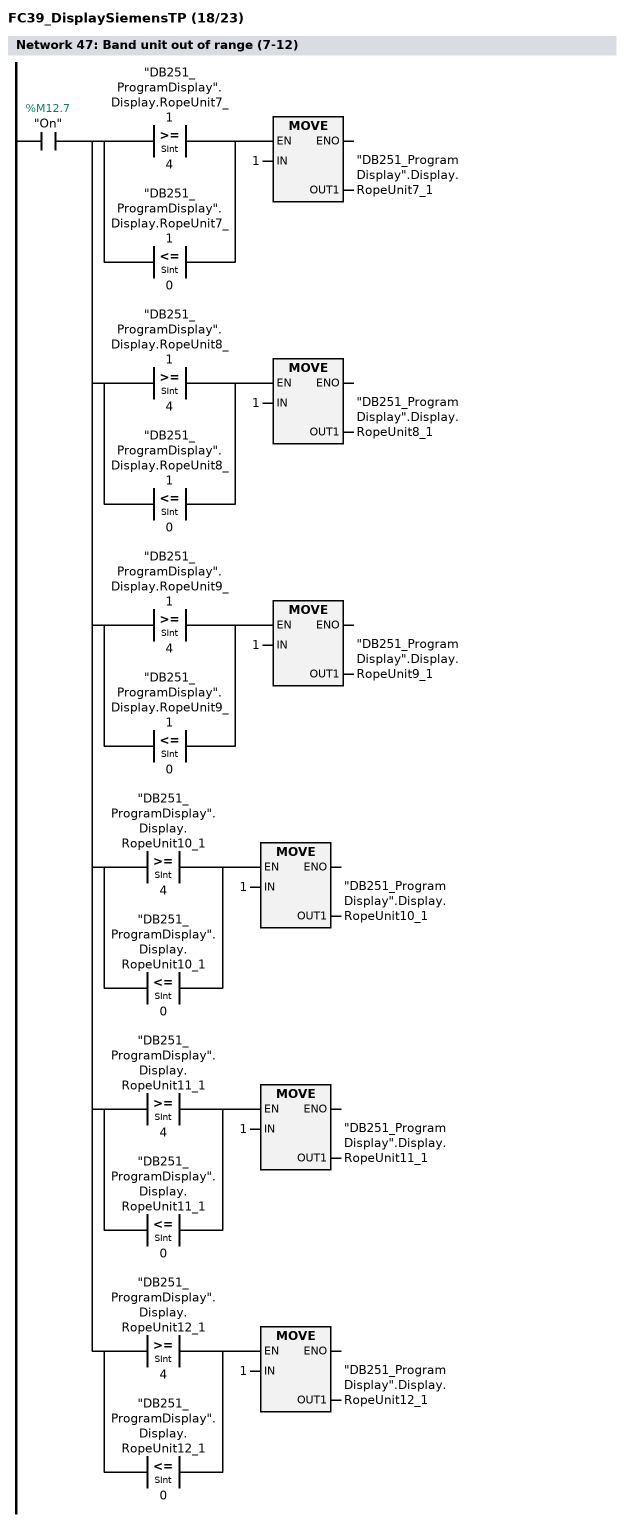
   RUNG wire#powerrail
      Contact( "On" )
      wire#w1
      { S7_Templates := "SrcType := SInt" } GE_Contact(in1 := "DB251_ProgramDisplay".Display.RopeUnit7_1, in2 := 4)
      wire#w2
      { S7_GenerateENO := "TRUE" } Move(in := 1, out1 => "DB251_ProgramDisplay".Display.RopeUnit7_1)
   END_RUNG
   RUNG wire#w1
      { S7_Templates := "SrcType := SInt" } LE_Contact(in1 := "DB251_ProgramDisplay".Display.RopeUnit7_1, in2 := 0)
   END_RUNG wire#w2
   RUNG wire#w1
      { S7_Templates := "SrcType := SInt" } GE_Contact(in1 := "DB251_ProgramDisplay".Display.RopeUnit8_1, in2 := 4)
      wire#w3
      { S7_GenerateENO := "TRUE" } Move(in := 1, out1 => "DB251_ProgramDisplay".Display.RopeUnit8_1)
   END_RUNG
   RUNG wire#w1
      { S7_Templates := "SrcType := SInt" } LE_Contact(in1 := "DB251_ProgramDisplay".Display.RopeUnit8_1, in2 := 0)
   END_RUNG wire#w3
   RUNG wire#w1
      { S7_Templates := "SrcType := SInt" } GE_Contact(in1 := "DB251_ProgramDisplay".Display.RopeUnit9_1, in2 := 4)
      wire#w4
      { S7_GenerateENO := "TRUE" } Move(in := 1, out1 => "DB251_ProgramDisplay".Display.RopeUnit9_1)
   END_RUNG
   RUNG wire#w1
      { S7_Templates := "SrcType := SInt" } LE_Contact(in1 := "DB251_ProgramDisplay".Display.RopeUnit9_1, in2 := 0)
   END_RUNG wire#w4
   RUNG wire#w1
      { S7_Templates := "SrcType := SInt" } GE_Contact(in1 := "DB251_ProgramDisplay".Display.RopeUnit10_1, in2 := 4)
      wire#w5
      { S7_GenerateENO := "TRUE" } Move(in := 1, out1 => "DB251_ProgramDisplay".Display.RopeUnit10_1)
   END_RUNG
   RUNG wire#w1
      { S7_Templates := "SrcType := SInt" } LE_Contact(in1 := "DB251_ProgramDisplay".Display.RopeUnit10_1, in2 := 0)
   END_RUNG wire#w5
   RUNG wire#w1
      { S7_Templates := "SrcType := SInt" } GE_Contact(in1 := "DB251_ProgramDisplay".Display.RopeUnit11_1, in2 := 4)
      wire#w6
      { S7_GenerateENO := "TRUE" } Move(in := 1, out1 => "DB251_ProgramDisplay".Display.RopeUnit11_1)
   END_RUNG
   RUNG wire#w1
      { S7_Templates := "SrcType := SInt" } LE_Contact(in1 := "DB251_ProgramDisplay".Display.RopeUnit11_1, in2 := 0)
   END_RUNG wire#w6
   RUNG wire#w1
      { S7_Templates := "SrcType := SInt" } GE_Contact(in1 := "DB251_ProgramDisplay".Display.RopeUnit12_1, in2 := 4)
      wire#w7
      { S7_GenerateENO := "TRUE" } Move(in := 1, out1 => "DB251_ProgramDisplay".Display.RopeUnit12_1)
   END_RUNG
   RUNG wire#w1
      { S7_Templates := "SrcType := SInt" } LE_Contact(in1 := "DB251_ProgramDisplay".Display.RopeUnit12_1, in2 := 0)
   END_RUNG wire#w7
   // the same network as SCL:
   IF "On" AND (("DB251_ProgramDisplay".Display.RopeUnit7_1 >= 4) OR ("DB251_ProgramDisplay".Display.RopeUnit7_1 <= 0)) THEN
       "DB251_ProgramDisplay".Display.RopeUnit7_1 := 1;
   END_IF;
   IF "On" AND (("DB251_ProgramDisplay".Display.RopeUnit8_1 >= 4) OR ("DB251_ProgramDisplay".Display.RopeUnit8_1 <= 0)) THEN
       "DB251_ProgramDisplay".Display.RopeUnit8_1 := 1;
   END_IF;
   IF "On" AND (("DB251_ProgramDisplay".Display.RopeUnit9_1 >= 4) OR ("DB251_ProgramDisplay".Display.RopeUnit9_1 <= 0)) THEN
       "DB251_ProgramDisplay".Display.RopeUnit9_1 := 1;
   END_IF;
   IF "On" AND (("DB251_ProgramDisplay".Display.RopeUnit10_1 >= 4) OR ("DB251_ProgramDisplay".Display.RopeUnit10_1 <= 0)) THEN
       "DB251_ProgramDisplay".Display.RopeUnit10_1 := 1;
   END_IF;
   IF "On" AND (("DB251_ProgramDisplay".Display.RopeUnit11_1 >= 4) OR ("DB251_ProgramDisplay".Display.RopeUnit11_1 <= 0)) THEN
       "DB251_ProgramDisplay".Display.RopeUnit11_1 := 1;
   END_IF;
   IF "On" AND (("DB251_ProgramDisplay".Display.RopeUnit12_1 >= 4) OR ("DB251_ProgramDisplay".Display.RopeUnit12_1 <= 0)) THEN
       "DB251_ProgramDisplay".Display.RopeUnit12_1 := 1;
   END_IF;
END_REGION

REGION Network 48: Rope unit out of range (1-6)
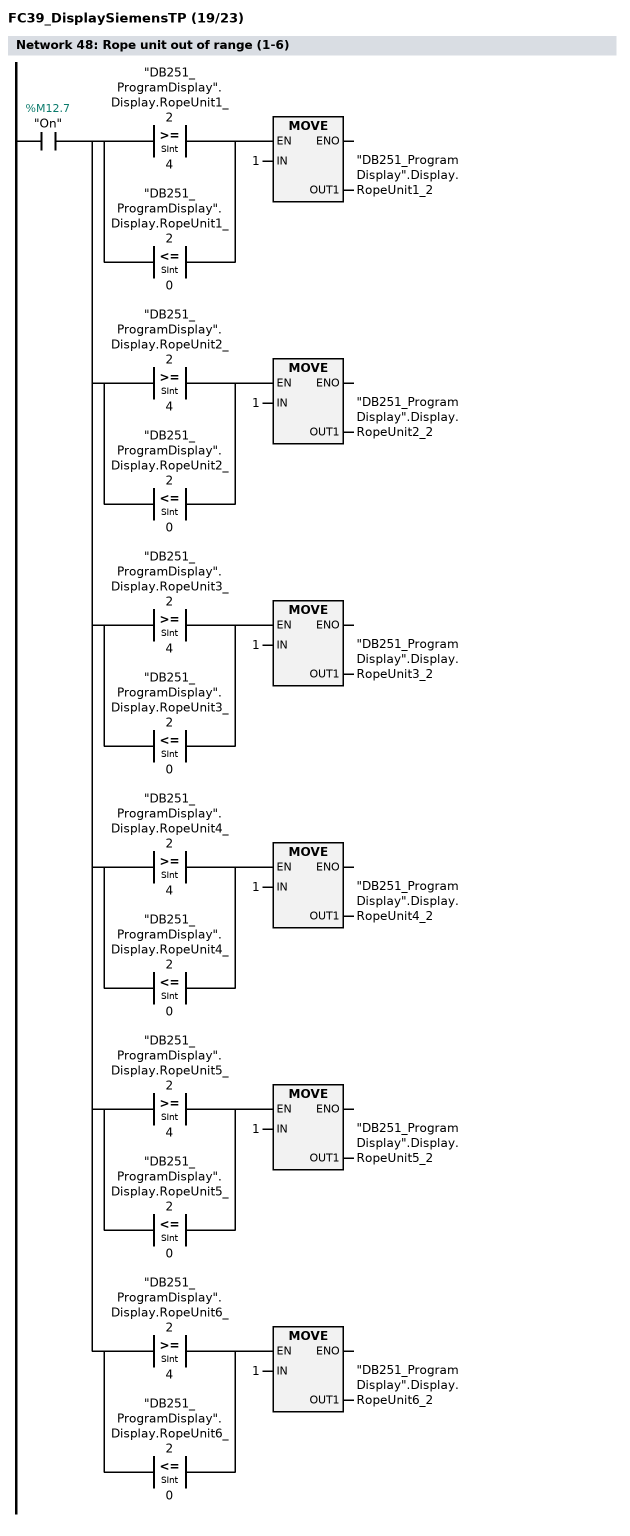
   RUNG wire#powerrail
      Contact( "On" )
      wire#w1
      { S7_Templates := "SrcType := SInt" } GE_Contact(in1 := "DB251_ProgramDisplay".Display.RopeUnit1_2, in2 := 4)
      wire#w2
      { S7_GenerateENO := "TRUE" } Move(in := 1, out1 => "DB251_ProgramDisplay".Display.RopeUnit1_2)
   END_RUNG
   RUNG wire#w1
      { S7_Templates := "SrcType := SInt" } LE_Contact(in1 := "DB251_ProgramDisplay".Display.RopeUnit1_2, in2 := 0)
   END_RUNG wire#w2
   RUNG wire#w1
      { S7_Templates := "SrcType := SInt" } GE_Contact(in1 := "DB251_ProgramDisplay".Display.RopeUnit2_2, in2 := 4)
      wire#w3
      { S7_GenerateENO := "TRUE" } Move(in := 1, out1 => "DB251_ProgramDisplay".Display.RopeUnit2_2)
   END_RUNG
   RUNG wire#w1
      { S7_Templates := "SrcType := SInt" } LE_Contact(in1 := "DB251_ProgramDisplay".Display.RopeUnit2_2, in2 := 0)
   END_RUNG wire#w3
   RUNG wire#w1
      { S7_Templates := "SrcType := SInt" } GE_Contact(in1 := "DB251_ProgramDisplay".Display.RopeUnit3_2, in2 := 4)
      wire#w4
      { S7_GenerateENO := "TRUE" } Move(in := 1, out1 => "DB251_ProgramDisplay".Display.RopeUnit3_2)
   END_RUNG
   RUNG wire#w1
      { S7_Templates := "SrcType := SInt" } LE_Contact(in1 := "DB251_ProgramDisplay".Display.RopeUnit3_2, in2 := 0)
   END_RUNG wire#w4
   RUNG wire#w1
      { S7_Templates := "SrcType := SInt" } GE_Contact(in1 := "DB251_ProgramDisplay".Display.RopeUnit4_2, in2 := 4)
      wire#w5
      { S7_GenerateENO := "TRUE" } Move(in := 1, out1 => "DB251_ProgramDisplay".Display.RopeUnit4_2)
   END_RUNG
   RUNG wire#w1
      { S7_Templates := "SrcType := SInt" } LE_Contact(in1 := "DB251_ProgramDisplay".Display.RopeUnit4_2, in2 := 0)
   END_RUNG wire#w5
   RUNG wire#w1
      { S7_Templates := "SrcType := SInt" } GE_Contact(in1 := "DB251_ProgramDisplay".Display.RopeUnit5_2, in2 := 4)
      wire#w6
      { S7_GenerateENO := "TRUE" } Move(in := 1, out1 => "DB251_ProgramDisplay".Display.RopeUnit5_2)
   END_RUNG
   RUNG wire#w1
      { S7_Templates := "SrcType := SInt" } LE_Contact(in1 := "DB251_ProgramDisplay".Display.RopeUnit5_2, in2 := 0)
   END_RUNG wire#w6
   RUNG wire#w1
      { S7_Templates := "SrcType := SInt" } GE_Contact(in1 := "DB251_ProgramDisplay".Display.RopeUnit6_2, in2 := 4)
      wire#w7
      { S7_GenerateENO := "TRUE" } Move(in := 1, out1 => "DB251_ProgramDisplay".Display.RopeUnit6_2)
   END_RUNG
   RUNG wire#w1
      { S7_Templates := "SrcType := SInt" } LE_Contact(in1 := "DB251_ProgramDisplay".Display.RopeUnit6_2, in2 := 0)
   END_RUNG wire#w7
   // the same network as SCL:
   IF "On" AND (("DB251_ProgramDisplay".Display.RopeUnit1_2 >= 4) OR ("DB251_ProgramDisplay".Display.RopeUnit1_2 <= 0)) THEN
       "DB251_ProgramDisplay".Display.RopeUnit1_2 := 1;
   END_IF;
   IF "On" AND (("DB251_ProgramDisplay".Display.RopeUnit2_2 >= 4) OR ("DB251_ProgramDisplay".Display.RopeUnit2_2 <= 0)) THEN
       "DB251_ProgramDisplay".Display.RopeUnit2_2 := 1;
   END_IF;
   IF "On" AND (("DB251_ProgramDisplay".Display.RopeUnit3_2 >= 4) OR ("DB251_ProgramDisplay".Display.RopeUnit3_2 <= 0)) THEN
       "DB251_ProgramDisplay".Display.RopeUnit3_2 := 1;
   END_IF;
   IF "On" AND (("DB251_ProgramDisplay".Display.RopeUnit4_2 >= 4) OR ("DB251_ProgramDisplay".Display.RopeUnit4_2 <= 0)) THEN
       "DB251_ProgramDisplay".Display.RopeUnit4_2 := 1;
   END_IF;
   IF "On" AND (("DB251_ProgramDisplay".Display.RopeUnit5_2 >= 4) OR ("DB251_ProgramDisplay".Display.RopeUnit5_2 <= 0)) THEN
       "DB251_ProgramDisplay".Display.RopeUnit5_2 := 1;
   END_IF;
   IF "On" AND (("DB251_ProgramDisplay".Display.RopeUnit6_2 >= 4) OR ("DB251_ProgramDisplay".Display.RopeUnit6_2 <= 0)) THEN
       "DB251_ProgramDisplay".Display.RopeUnit6_2 := 1;
   END_IF;
END_REGION

REGION Network 49: Rope unit out of range (7-12)
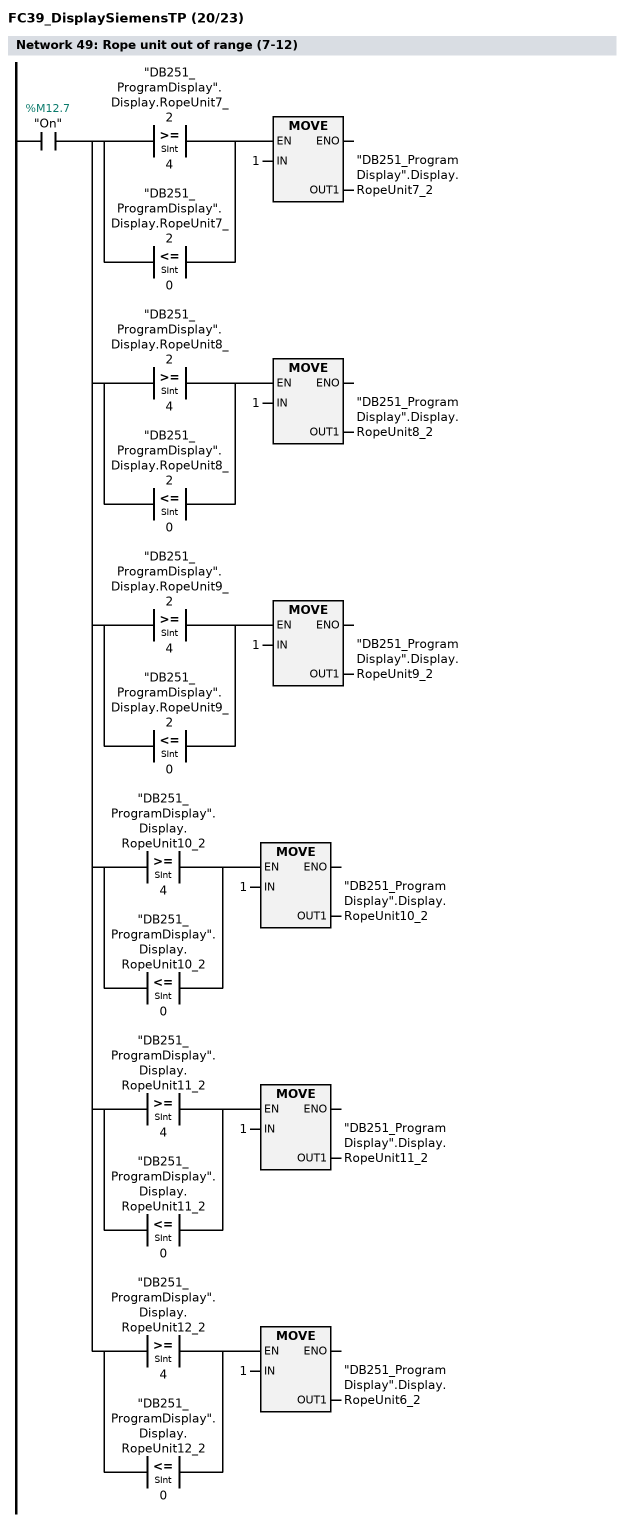
   RUNG wire#powerrail
      Contact( "On" )
      wire#w1
      { S7_Templates := "SrcType := SInt" } GE_Contact(in1 := "DB251_ProgramDisplay".Display.RopeUnit7_2, in2 := 4)
      wire#w2
      { S7_GenerateENO := "TRUE" } Move(in := 1, out1 => "DB251_ProgramDisplay".Display.RopeUnit7_2)
   END_RUNG
   RUNG wire#w1
      { S7_Templates := "SrcType := SInt" } LE_Contact(in1 := "DB251_ProgramDisplay".Display.RopeUnit7_2, in2 := 0)
   END_RUNG wire#w2
   RUNG wire#w1
      { S7_Templates := "SrcType := SInt" } GE_Contact(in1 := "DB251_ProgramDisplay".Display.RopeUnit8_2, in2 := 4)
      wire#w3
      { S7_GenerateENO := "TRUE" } Move(in := 1, out1 => "DB251_ProgramDisplay".Display.RopeUnit8_2)
   END_RUNG
   RUNG wire#w1
      { S7_Templates := "SrcType := SInt" } LE_Contact(in1 := "DB251_ProgramDisplay".Display.RopeUnit8_2, in2 := 0)
   END_RUNG wire#w3
   RUNG wire#w1
      { S7_Templates := "SrcType := SInt" } GE_Contact(in1 := "DB251_ProgramDisplay".Display.RopeUnit9_2, in2 := 4)
      wire#w4
      { S7_GenerateENO := "TRUE" } Move(in := 1, out1 => "DB251_ProgramDisplay".Display.RopeUnit9_2)
   END_RUNG
   RUNG wire#w1
      { S7_Templates := "SrcType := SInt" } LE_Contact(in1 := "DB251_ProgramDisplay".Display.RopeUnit9_2, in2 := 0)
   END_RUNG wire#w4
   RUNG wire#w1
      { S7_Templates := "SrcType := SInt" } GE_Contact(in1 := "DB251_ProgramDisplay".Display.RopeUnit10_2, in2 := 4)
      wire#w5
      { S7_GenerateENO := "TRUE" } Move(in := 1, out1 => "DB251_ProgramDisplay".Display.RopeUnit10_2)
   END_RUNG
   RUNG wire#w1
      { S7_Templates := "SrcType := SInt" } LE_Contact(in1 := "DB251_ProgramDisplay".Display.RopeUnit10_2, in2 := 0)
   END_RUNG wire#w5
   RUNG wire#w1
      { S7_Templates := "SrcType := SInt" } GE_Contact(in1 := "DB251_ProgramDisplay".Display.RopeUnit11_2, in2 := 4)
      wire#w6
      { S7_GenerateENO := "TRUE" } Move(in := 1, out1 => "DB251_ProgramDisplay".Display.RopeUnit11_2)
   END_RUNG
   RUNG wire#w1
      { S7_Templates := "SrcType := SInt" } LE_Contact(in1 := "DB251_ProgramDisplay".Display.RopeUnit11_2, in2 := 0)
   END_RUNG wire#w6
   RUNG wire#w1
      { S7_Templates := "SrcType := SInt" } GE_Contact(in1 := "DB251_ProgramDisplay".Display.RopeUnit12_2, in2 := 4)
      wire#w7
      { S7_GenerateENO := "TRUE" } Move(in := 1, out1 => "DB251_ProgramDisplay".Display.RopeUnit6_2)
   END_RUNG
   RUNG wire#w1
      { S7_Templates := "SrcType := SInt" } LE_Contact(in1 := "DB251_ProgramDisplay".Display.RopeUnit12_2, in2 := 0)
   END_RUNG wire#w7
   // the same network as SCL:
   IF "On" AND (("DB251_ProgramDisplay".Display.RopeUnit7_2 >= 4) OR ("DB251_ProgramDisplay".Display.RopeUnit7_2 <= 0)) THEN
       "DB251_ProgramDisplay".Display.RopeUnit7_2 := 1;
   END_IF;
   IF "On" AND (("DB251_ProgramDisplay".Display.RopeUnit8_2 >= 4) OR ("DB251_ProgramDisplay".Display.RopeUnit8_2 <= 0)) THEN
       "DB251_ProgramDisplay".Display.RopeUnit8_2 := 1;
   END_IF;
   IF "On" AND (("DB251_ProgramDisplay".Display.RopeUnit9_2 >= 4) OR ("DB251_ProgramDisplay".Display.RopeUnit9_2 <= 0)) THEN
       "DB251_ProgramDisplay".Display.RopeUnit9_2 := 1;
   END_IF;
   IF "On" AND (("DB251_ProgramDisplay".Display.RopeUnit10_2 >= 4) OR ("DB251_ProgramDisplay".Display.RopeUnit10_2 <= 0)) THEN
       "DB251_ProgramDisplay".Display.RopeUnit10_2 := 1;
   END_IF;
   IF "On" AND (("DB251_ProgramDisplay".Display.RopeUnit11_2 >= 4) OR ("DB251_ProgramDisplay".Display.RopeUnit11_2 <= 0)) THEN
       "DB251_ProgramDisplay".Display.RopeUnit11_2 := 1;
   END_IF;
   IF "On" AND (("DB251_ProgramDisplay".Display.RopeUnit12_2 >= 4) OR ("DB251_ProgramDisplay".Display.RopeUnit12_2 <= 0)) THEN
       "DB251_ProgramDisplay".Display.RopeUnit6_2 := 1;
   END_IF;
END_REGION

REGION Network 50: Define landmark to bottom for the last step
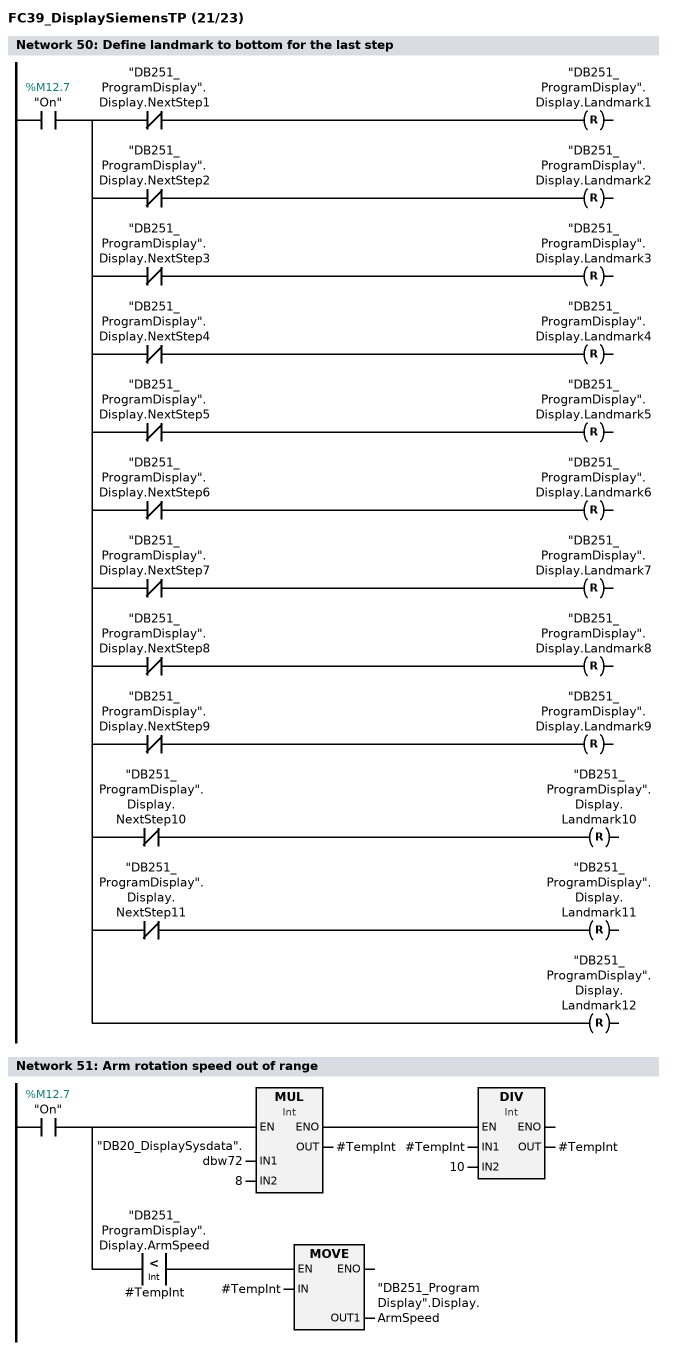
   RUNG wire#powerrail
      Contact( "On" )
      wire#w1
      I_Contact( "DB251_ProgramDisplay".Display.NextStep1 )
      R_Coil( "DB251_ProgramDisplay".Display.Landmark1 )
   END_RUNG
   RUNG wire#w1
      I_Contact( "DB251_ProgramDisplay".Display.NextStep2 )
      R_Coil( "DB251_ProgramDisplay".Display.Landmark2 )
   END_RUNG
   RUNG wire#w1
      I_Contact( "DB251_ProgramDisplay".Display.NextStep3 )
      R_Coil( "DB251_ProgramDisplay".Display.Landmark3 )
   END_RUNG
   RUNG wire#w1
      I_Contact( "DB251_ProgramDisplay".Display.NextStep4 )
      R_Coil( "DB251_ProgramDisplay".Display.Landmark4 )
   END_RUNG
   RUNG wire#w1
      I_Contact( "DB251_ProgramDisplay".Display.NextStep5 )
      R_Coil( "DB251_ProgramDisplay".Display.Landmark5 )
   END_RUNG
   RUNG wire#w1
      I_Contact( "DB251_ProgramDisplay".Display.NextStep6 )
      R_Coil( "DB251_ProgramDisplay".Display.Landmark6 )
   END_RUNG
   RUNG wire#w1
      I_Contact( "DB251_ProgramDisplay".Display.NextStep7 )
      R_Coil( "DB251_ProgramDisplay".Display.Landmark7 )
   END_RUNG
   RUNG wire#w1
      I_Contact( "DB251_ProgramDisplay".Display.NextStep8 )
      R_Coil( "DB251_ProgramDisplay".Display.Landmark8 )
   END_RUNG
   RUNG wire#w1
      I_Contact( "DB251_ProgramDisplay".Display.NextStep9 )
      R_Coil( "DB251_ProgramDisplay".Display.Landmark9 )
   END_RUNG
   RUNG wire#w1
      I_Contact( "DB251_ProgramDisplay".Display.NextStep10 )
      R_Coil( "DB251_ProgramDisplay".Display.Landmark10 )
   END_RUNG
   RUNG wire#w1
      I_Contact( "DB251_ProgramDisplay".Display.NextStep11 )
      R_Coil( "DB251_ProgramDisplay".Display.Landmark11 )
   END_RUNG
   RUNG wire#w1
      R_Coil( "DB251_ProgramDisplay".Display.Landmark12 )
   END_RUNG
   // the same network as SCL:
   IF "On" AND NOT "DB251_ProgramDisplay".Display.NextStep1 THEN
       "DB251_ProgramDisplay".Display.Landmark1 := FALSE;
   END_IF;
   IF "On" AND NOT "DB251_ProgramDisplay".Display.NextStep2 THEN
       "DB251_ProgramDisplay".Display.Landmark2 := FALSE;
   END_IF;
   IF "On" AND NOT "DB251_ProgramDisplay".Display.NextStep3 THEN
       "DB251_ProgramDisplay".Display.Landmark3 := FALSE;
   END_IF;
   IF "On" AND NOT "DB251_ProgramDisplay".Display.NextStep4 THEN
       "DB251_ProgramDisplay".Display.Landmark4 := FALSE;
   END_IF;
   IF "On" AND NOT "DB251_ProgramDisplay".Display.NextStep5 THEN
       "DB251_ProgramDisplay".Display.Landmark5 := FALSE;
   END_IF;
   IF "On" AND NOT "DB251_ProgramDisplay".Display.NextStep6 THEN
       "DB251_ProgramDisplay".Display.Landmark6 := FALSE;
   END_IF;
   IF "On" AND NOT "DB251_ProgramDisplay".Display.NextStep7 THEN
       "DB251_ProgramDisplay".Display.Landmark7 := FALSE;
   END_IF;
   IF "On" AND NOT "DB251_ProgramDisplay".Display.NextStep8 THEN
       "DB251_ProgramDisplay".Display.Landmark8 := FALSE;
   END_IF;
   IF "On" AND NOT "DB251_ProgramDisplay".Display.NextStep9 THEN
       "DB251_ProgramDisplay".Display.Landmark9 := FALSE;
   END_IF;
   IF "On" AND NOT "DB251_ProgramDisplay".Display.NextStep10 THEN
       "DB251_ProgramDisplay".Display.Landmark10 := FALSE;
   END_IF;
   IF "On" AND NOT "DB251_ProgramDisplay".Display.NextStep11 THEN
       "DB251_ProgramDisplay".Display.Landmark11 := FALSE;
   END_IF;
   IF "On" THEN "DB251_ProgramDisplay".Display.Landmark12 := FALSE; END_IF;
END_REGION

REGION Network 51: Arm rotation speed out of range
   RUNG wire#powerrail
      Contact( "On" )
      wire#w1
      { S7_Templates := "SrcType := Int"; S7_GenerateENO := "TRUE" } Mul(in1 := "DB20_DisplaySysdata".dbw72, in2 := 8, out => #TempInt)
      { S7_Templates := "SrcType := Int"; S7_GenerateENO := "TRUE" } Div(in1 := #TempInt, in2 := 10, out => #TempInt)
   END_RUNG
   RUNG wire#w1
      { S7_Templates := "SrcType := Int" } LT_Contact(in1 := "DB251_ProgramDisplay".Display.ArmSpeed, in2 := #TempInt)
      { S7_GenerateENO := "TRUE" } Move(in := #TempInt, out1 => "DB251_ProgramDisplay".Display.ArmSpeed)
   END_RUNG
   // the same network as SCL:
   // ENO of a box is taken as its EN; it also drops when the box reports an error
   IF "On" THEN
       #TempInt := "DB20_DisplaySysdata".dbw72 * 8;
       #TempInt := #TempInt / 10;
   END_IF;
   IF "On" AND ("DB251_ProgramDisplay".Display.ArmSpeed < #TempInt) THEN
       "DB251_ProgramDisplay".Display.ArmSpeed := #TempInt;
   END_IF;
END_REGION

REGION Network 52: Next step for spool carriage height 12 (0=End 1=Next)
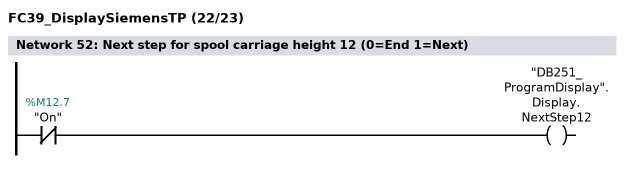
   RUNG wire#powerrail
      I_Contact( "On" )
      Coil( "DB251_ProgramDisplay".Display.NextStep12 )
   END_RUNG
   // the same network as SCL:
   "DB251_ProgramDisplay".Display.NextStep12 := NOT "On";
END_REGION

REGION Network 53
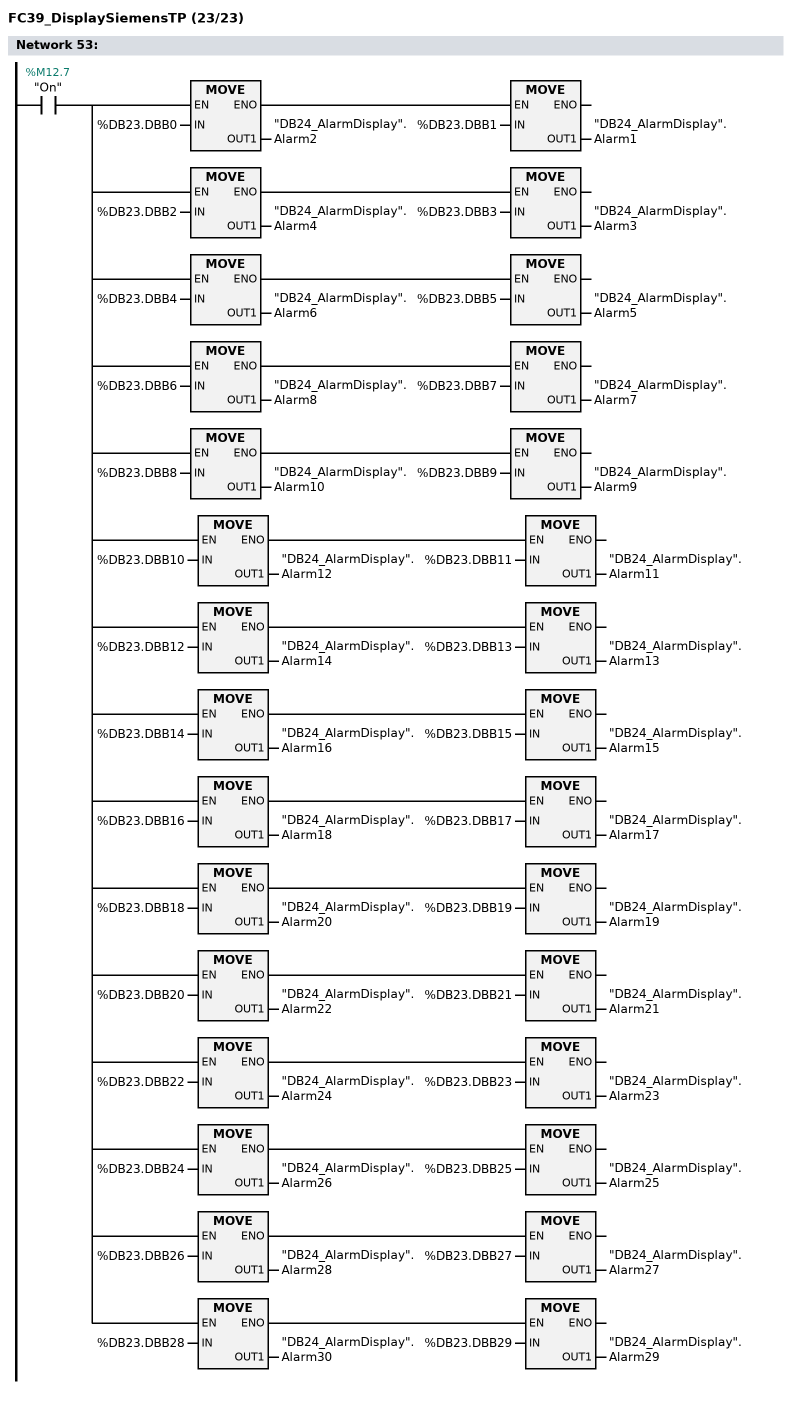
   RUNG wire#powerrail
      Contact( "On" )
      wire#w1
      { S7_GenerateENO := "TRUE" } Move(in := %DB23.DBB0, out1 => "DB24_AlarmDisplay".Alarm2)
      { S7_GenerateENO := "TRUE" } Move(in := %DB23.DBB1, out1 => "DB24_AlarmDisplay".Alarm1)
   END_RUNG
   RUNG wire#w1
      { S7_GenerateENO := "TRUE" } Move(in := %DB23.DBB2, out1 => "DB24_AlarmDisplay".Alarm4)
      { S7_GenerateENO := "TRUE" } Move(in := %DB23.DBB3, out1 => "DB24_AlarmDisplay".Alarm3)
   END_RUNG
   RUNG wire#w1
      { S7_GenerateENO := "TRUE" } Move(in := %DB23.DBB4, out1 => "DB24_AlarmDisplay".Alarm6)
      { S7_GenerateENO := "TRUE" } Move(in := %DB23.DBB5, out1 => "DB24_AlarmDisplay".Alarm5)
   END_RUNG
   RUNG wire#w1
      { S7_GenerateENO := "TRUE" } Move(in := %DB23.DBB6, out1 => "DB24_AlarmDisplay".Alarm8)
      { S7_GenerateENO := "TRUE" } Move(in := %DB23.DBB7, out1 => "DB24_AlarmDisplay".Alarm7)
   END_RUNG
   RUNG wire#w1
      { S7_GenerateENO := "TRUE" } Move(in := %DB23.DBB8, out1 => "DB24_AlarmDisplay".Alarm10)
      { S7_GenerateENO := "TRUE" } Move(in := %DB23.DBB9, out1 => "DB24_AlarmDisplay".Alarm9)
   END_RUNG
   RUNG wire#w1
      { S7_GenerateENO := "TRUE" } Move(in := %DB23.DBB10, out1 => "DB24_AlarmDisplay".Alarm12)
      { S7_GenerateENO := "TRUE" } Move(in := %DB23.DBB11, out1 => "DB24_AlarmDisplay".Alarm11)
   END_RUNG
   RUNG wire#w1
      { S7_GenerateENO := "TRUE" } Move(in := %DB23.DBB12, out1 => "DB24_AlarmDisplay".Alarm14)
      { S7_GenerateENO := "TRUE" } Move(in := %DB23.DBB13, out1 => "DB24_AlarmDisplay".Alarm13)
   END_RUNG
   RUNG wire#w1
      { S7_GenerateENO := "TRUE" } Move(in := %DB23.DBB14, out1 => "DB24_AlarmDisplay".Alarm16)
      { S7_GenerateENO := "TRUE" } Move(in := %DB23.DBB15, out1 => "DB24_AlarmDisplay".Alarm15)
   END_RUNG
   RUNG wire#w1
      { S7_GenerateENO := "TRUE" } Move(in := %DB23.DBB16, out1 => "DB24_AlarmDisplay".Alarm18)
      { S7_GenerateENO := "TRUE" } Move(in := %DB23.DBB17, out1 => "DB24_AlarmDisplay".Alarm17)
   END_RUNG
   RUNG wire#w1
      { S7_GenerateENO := "TRUE" } Move(in := %DB23.DBB18, out1 => "DB24_AlarmDisplay".Alarm20)
      { S7_GenerateENO := "TRUE" } Move(in := %DB23.DBB19, out1 => "DB24_AlarmDisplay".Alarm19)
   END_RUNG
   RUNG wire#w1
      { S7_GenerateENO := "TRUE" } Move(in := %DB23.DBB20, out1 => "DB24_AlarmDisplay".Alarm22)
      { S7_GenerateENO := "TRUE" } Move(in := %DB23.DBB21, out1 => "DB24_AlarmDisplay".Alarm21)
   END_RUNG
   RUNG wire#w1
      { S7_GenerateENO := "TRUE" } Move(in := %DB23.DBB22, out1 => "DB24_AlarmDisplay".Alarm24)
      { S7_GenerateENO := "TRUE" } Move(in := %DB23.DBB23, out1 => "DB24_AlarmDisplay".Alarm23)
   END_RUNG
   RUNG wire#w1
      { S7_GenerateENO := "TRUE" } Move(in := %DB23.DBB24, out1 => "DB24_AlarmDisplay".Alarm26)
      { S7_GenerateENO := "TRUE" } Move(in := %DB23.DBB25, out1 => "DB24_AlarmDisplay".Alarm25)
   END_RUNG
   RUNG wire#w1
      { S7_GenerateENO := "TRUE" } Move(in := %DB23.DBB26, out1 => "DB24_AlarmDisplay".Alarm28)
      { S7_GenerateENO := "TRUE" } Move(in := %DB23.DBB27, out1 => "DB24_AlarmDisplay".Alarm27)
   END_RUNG
   RUNG wire#w1
      { S7_GenerateENO := "TRUE" } Move(in := %DB23.DBB28, out1 => "DB24_AlarmDisplay".Alarm30)
      { S7_GenerateENO := "TRUE" } Move(in := %DB23.DBB29, out1 => "DB24_AlarmDisplay".Alarm29)
   END_RUNG
   // the same network as SCL:
   // ENO of a box is taken as its EN; it also drops when the box reports an error
   IF "On" THEN
       "DB24_AlarmDisplay".Alarm2 := %DB23.DBB0;
       "DB24_AlarmDisplay".Alarm1 := %DB23.DBB1;
       "DB24_AlarmDisplay".Alarm4 := %DB23.DBB2;
       "DB24_AlarmDisplay".Alarm3 := %DB23.DBB3;
       "DB24_AlarmDisplay".Alarm6 := %DB23.DBB4;
       "DB24_AlarmDisplay".Alarm5 := %DB23.DBB5;
       "DB24_AlarmDisplay".Alarm8 := %DB23.DBB6;
       "DB24_AlarmDisplay".Alarm7 := %DB23.DBB7;
       "DB24_AlarmDisplay".Alarm10 := %DB23.DBB8;
       "DB24_AlarmDisplay".Alarm9 := %DB23.DBB9;
       "DB24_AlarmDisplay".Alarm12 := %DB23.DBB10;
       "DB24_AlarmDisplay".Alarm11 := %DB23.DBB11;
       "DB24_AlarmDisplay".Alarm14 := %DB23.DBB12;
       "DB24_AlarmDisplay".Alarm13 := %DB23.DBB13;
       "DB24_AlarmDisplay".Alarm16 := %DB23.DBB14;
       "DB24_AlarmDisplay".Alarm15 := %DB23.DBB15;
       "DB24_AlarmDisplay".Alarm18 := %DB23.DBB16;
       "DB24_AlarmDisplay".Alarm17 := %DB23.DBB17;
       "DB24_AlarmDisplay".Alarm20 := %DB23.DBB18;
       "DB24_AlarmDisplay".Alarm19 := %DB23.DBB19;
       "DB24_AlarmDisplay".Alarm22 := %DB23.DBB20;
       "DB24_AlarmDisplay".Alarm21 := %DB23.DBB21;
       "DB24_AlarmDisplay".Alarm24 := %DB23.DBB22;
       "DB24_AlarmDisplay".Alarm23 := %DB23.DBB23;
       "DB24_AlarmDisplay".Alarm26 := %DB23.DBB24;
       "DB24_AlarmDisplay".Alarm25 := %DB23.DBB25;
       "DB24_AlarmDisplay".Alarm28 := %DB23.DBB26;
       "DB24_AlarmDisplay".Alarm27 := %DB23.DBB27;
       "DB24_AlarmDisplay".Alarm30 := %DB23.DBB28;
       "DB24_AlarmDisplay".Alarm29 := %DB23.DBB29;
   END_IF;
END_REGION
END_FUNCTION

FUNCTION "FC105_GreyBarReset" : Void   // FC105, LAD
TITLE = Reset grey bar program data
{ S7_Optimized_Access := 'TRUE' }
VERSION : 0.1
// stored: AutoNumber false, IsIECCheckEnabled false, SetENOAutomatically false, UDAEnableTagReadback false
BEGIN

REGION Network 1: Reset grey bar program data
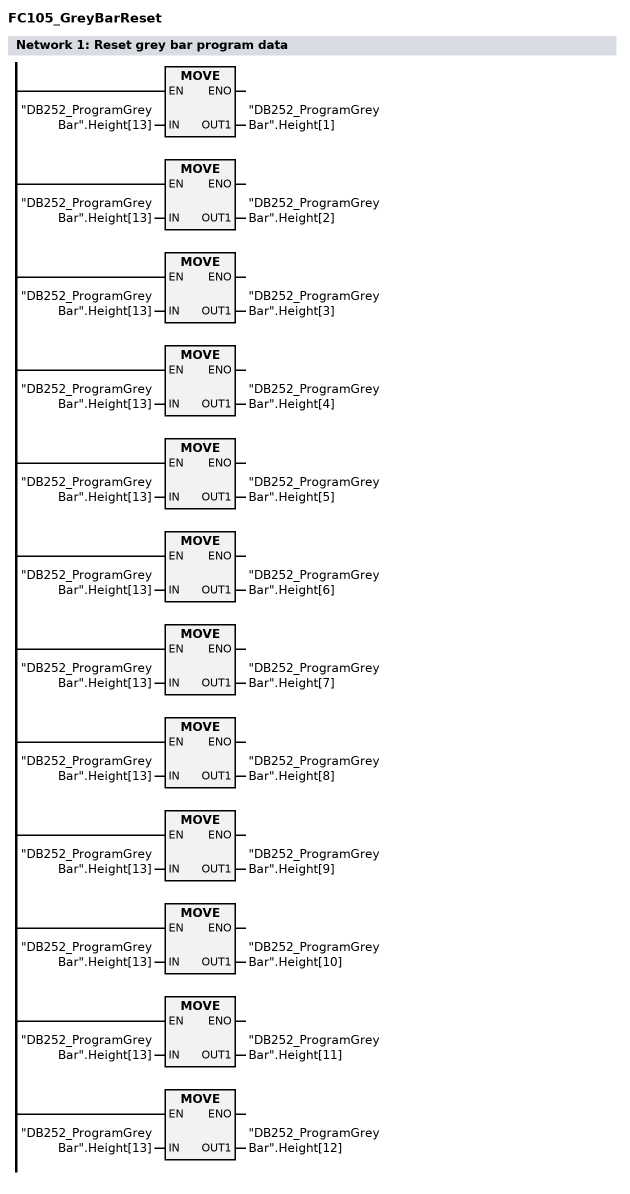
   RUNG wire#powerrail
      { S7_GenerateENO := "TRUE" } Move(in := "DB252_ProgramGreyBar".Height[13], out1 => "DB252_ProgramGreyBar".Height[1])
   END_RUNG
   RUNG wire#powerrail
      { S7_GenerateENO := "TRUE" } Move(in := "DB252_ProgramGreyBar".Height[13], out1 => "DB252_ProgramGreyBar".Height[2])
   END_RUNG
   RUNG wire#powerrail
      { S7_GenerateENO := "TRUE" } Move(in := "DB252_ProgramGreyBar".Height[13], out1 => "DB252_ProgramGreyBar".Height[3])
   END_RUNG
   RUNG wire#powerrail
      { S7_GenerateENO := "TRUE" } Move(in := "DB252_ProgramGreyBar".Height[13], out1 => "DB252_ProgramGreyBar".Height[4])
   END_RUNG
   RUNG wire#powerrail
      { S7_GenerateENO := "TRUE" } Move(in := "DB252_ProgramGreyBar".Height[13], out1 => "DB252_ProgramGreyBar".Height[5])
   END_RUNG
   RUNG wire#powerrail
      { S7_GenerateENO := "TRUE" } Move(in := "DB252_ProgramGreyBar".Height[13], out1 => "DB252_ProgramGreyBar".Height[6])
   END_RUNG
   RUNG wire#powerrail
      { S7_GenerateENO := "TRUE" } Move(in := "DB252_ProgramGreyBar".Height[13], out1 => "DB252_ProgramGreyBar".Height[7])
   END_RUNG
   RUNG wire#powerrail
      { S7_GenerateENO := "TRUE" } Move(in := "DB252_ProgramGreyBar".Height[13], out1 => "DB252_ProgramGreyBar".Height[8])
   END_RUNG
   RUNG wire#powerrail
      { S7_GenerateENO := "TRUE" } Move(in := "DB252_ProgramGreyBar".Height[13], out1 => "DB252_ProgramGreyBar".Height[9])
   END_RUNG
   RUNG wire#powerrail
      { S7_GenerateENO := "TRUE" } Move(in := "DB252_ProgramGreyBar".Height[13], out1 => "DB252_ProgramGreyBar".Height[10])
   END_RUNG
   RUNG wire#powerrail
      { S7_GenerateENO := "TRUE" } Move(in := "DB252_ProgramGreyBar".Height[13], out1 => "DB252_ProgramGreyBar".Height[11])
   END_RUNG
   RUNG wire#powerrail
      { S7_GenerateENO := "TRUE" } Move(in := "DB252_ProgramGreyBar".Height[13], out1 => "DB252_ProgramGreyBar".Height[12])
   END_RUNG
   // the same network as SCL:
   "DB252_ProgramGreyBar".Height[1] := "DB252_ProgramGreyBar".Height[13];
   "DB252_ProgramGreyBar".Height[2] := "DB252_ProgramGreyBar".Height[13];
   "DB252_ProgramGreyBar".Height[3] := "DB252_ProgramGreyBar".Height[13];
   "DB252_ProgramGreyBar".Height[4] := "DB252_ProgramGreyBar".Height[13];
   "DB252_ProgramGreyBar".Height[5] := "DB252_ProgramGreyBar".Height[13];
   "DB252_ProgramGreyBar".Height[6] := "DB252_ProgramGreyBar".Height[13];
   "DB252_ProgramGreyBar".Height[7] := "DB252_ProgramGreyBar".Height[13];
   "DB252_ProgramGreyBar".Height[8] := "DB252_ProgramGreyBar".Height[13];
   "DB252_ProgramGreyBar".Height[9] := "DB252_ProgramGreyBar".Height[13];
   "DB252_ProgramGreyBar".Height[10] := "DB252_ProgramGreyBar".Height[13];
   "DB252_ProgramGreyBar".Height[11] := "DB252_ProgramGreyBar".Height[13];
   "DB252_ProgramGreyBar".Height[12] := "DB252_ProgramGreyBar".Height[13];
END_REGION
END_FUNCTION

FUNCTION "FC41_NoRopeUnit" : Void   // FC41, LAD
TITLE = No rope unit
{ S7_Optimized_Access := 'FALSE' }
AUTHOR : Robopac
VERSION : 0.0
// stored: AutoNumber false, IsIECCheckEnabled false, SetENOAutomatically false, UDAEnableTagReadback false
BEGIN

REGION Network 1: RopeUnitOk1: Rope unit open
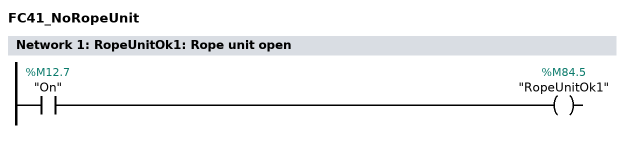
   RUNG wire#powerrail
      Contact( "On" )
      Coil( "RopeUnitOk1" )
   END_RUNG
   // the same network as SCL:
   "RopeUnitOk1" := "On";
END_REGION
END_FUNCTION

FUNCTION "FC42_RopeUnit" : Void   // FC42, LAD
TITLE = RopeUnit
{ S7_Optimized_Access := 'FALSE' }
VERSION : 0.1
// stored: AutoNumber false, IsIECCheckEnabled false, SetENOAutomatically false, UDAEnableTagReadback false
   VAR_TEMP
      OpenCloseDoubleRope : Bool;
      DoubleRopeOpen : Bool;
      TempInt : Int;
      TempInt1 : Int;
   END_VAR
   VAR_TEMP   // added for the SCL form of the ladder/FBD networks
      _w1 : Bool;
   END_VAR
BEGIN

REGION Network 1: Timeout for single or lower(double) rope unit open/close
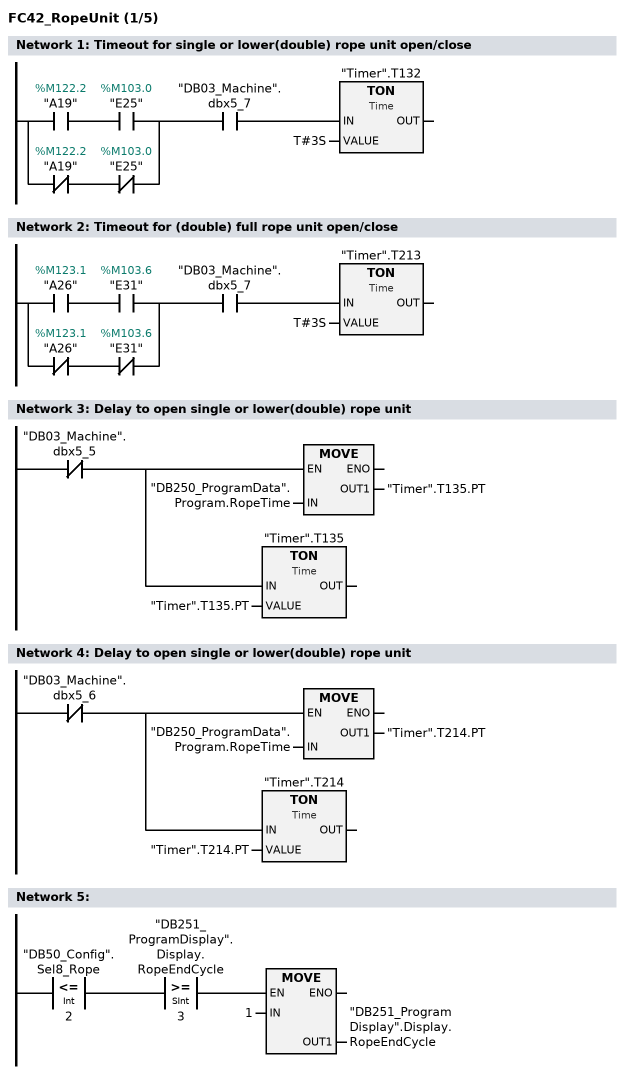
   "Timer".T132.TON(IN := (("A19" AND "E25") OR (NOT "A19" AND NOT "E25")) AND "DB03_Machine".dbx5_7, PT := T#3S);   // TON coil
END_REGION

REGION Network 2: Timeout for (double) full rope unit open/close
   "Timer".T213.TON(IN := (("A26" AND "E31") OR (NOT "A26" AND NOT "E31")) AND "DB03_Machine".dbx5_7, PT := T#3S);   // TON coil
END_REGION

REGION Network 3: Delay to open single or lower(double) rope unit
   #_w1 := NOT "DB03_Machine".dbx5_5;
   IF #_w1 THEN "Timer".T135.PT := "DB250_ProgramData".Program.RopeTime; END_IF;
   "Timer".T135.TON(IN := #_w1, PT := "Timer".T135.PT);   // TON coil
END_REGION

REGION Network 4: Delay to open single or lower(double) rope unit
   #_w1 := NOT "DB03_Machine".dbx5_6;
   IF #_w1 THEN "Timer".T214.PT := "DB250_ProgramData".Program.RopeTime; END_IF;
   "Timer".T214.TON(IN := #_w1, PT := "Timer".T214.PT);   // TON coil
END_REGION

REGION Network 5
   RUNG wire#powerrail
      { S7_Templates := "SrcType := Int" } LE_Contact(in1 := "DB50_Config".Sel8_Rope, in2 := 2)
      { S7_Templates := "SrcType := SInt" } GE_Contact(in1 := "DB251_ProgramDisplay".Display.RopeEndCycle, in2 := 3)
      { S7_GenerateENO := "TRUE" } Move(in := 1, out1 => "DB251_ProgramDisplay".Display.RopeEndCycle)
   END_RUNG
   // the same network as SCL:
   IF ("DB50_Config".Sel8_Rope <= 2) AND ("DB251_ProgramDisplay".Display.RopeEndCycle >= 3) THEN
       "DB251_ProgramDisplay".Display.RopeEndCycle := 1;
   END_IF;
END_REGION

REGION Network 6: RopeUnitOk1: Rope unit open
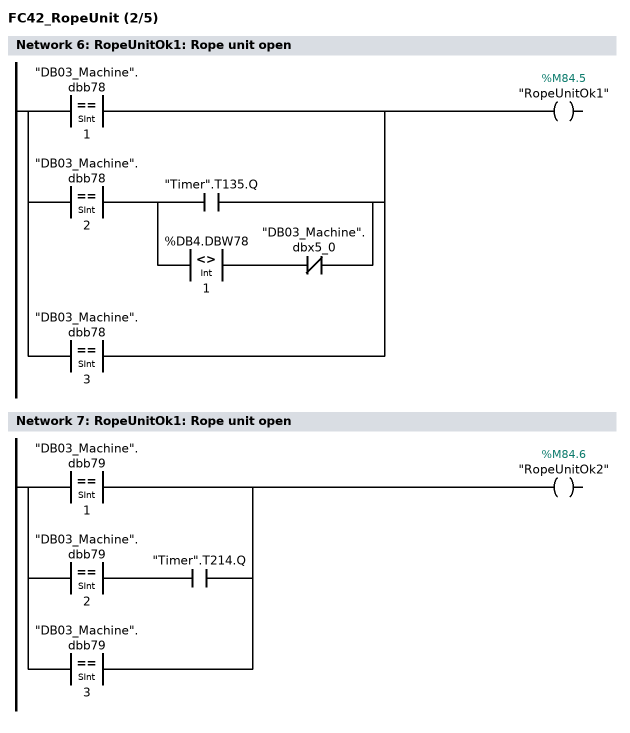
   RUNG wire#powerrail
      { S7_Templates := "SrcType := SInt" } EQ_Contact(in1 := "DB03_Machine".dbb78, in2 := 1)
      wire#w1
      Coil( "RopeUnitOk1" )
   END_RUNG
   RUNG wire#powerrail
      { S7_Templates := "SrcType := SInt" } EQ_Contact(in1 := "DB03_Machine".dbb78, in2 := 2)
      wire#w2
      Contact( "Timer".T135.Q )
   END_RUNG wire#w1
   RUNG wire#w2
      { S7_Templates := "SrcType := Int" } NE_Contact(in1 := %DB4.DBW78, in2 := 1)
      I_Contact( "DB03_Machine".dbx5_0 )
   END_RUNG wire#w1
   RUNG wire#powerrail
      { S7_Templates := "SrcType := SInt" } EQ_Contact(in1 := "DB03_Machine".dbb78, in2 := 3)
   END_RUNG wire#w1
   // the same network as SCL:
   "RopeUnitOk1" := ("DB03_Machine".dbb78 = 1) OR (("DB03_Machine".dbb78 = 2) AND ("Timer".T135.Q OR ((%DB4.DBW78 <> 1) AND NOT "DB03_Machine".dbx5_0))) OR ("DB03_Machine".dbb78 = 3);
END_REGION

REGION Network 7: RopeUnitOk1: Rope unit open
   RUNG wire#powerrail
      { S7_Templates := "SrcType := SInt" } EQ_Contact(in1 := "DB03_Machine".dbb79, in2 := 1)
      wire#w1
      Coil( "RopeUnitOk2" )
   END_RUNG
   RUNG wire#powerrail
      { S7_Templates := "SrcType := SInt" } EQ_Contact(in1 := "DB03_Machine".dbb79, in2 := 2)
      Contact( "Timer".T214.Q )
   END_RUNG wire#w1
   RUNG wire#powerrail
      { S7_Templates := "SrcType := SInt" } EQ_Contact(in1 := "DB03_Machine".dbb79, in2 := 3)
   END_RUNG wire#w1
   // the same network as SCL:
   "RopeUnitOk2" := ("DB03_Machine".dbb79 = 1) OR (("DB03_Machine".dbb79 = 2) AND "Timer".T214.Q) OR ("DB03_Machine".dbb79 = 3);
END_REGION

REGION Network 8: Closing upper(double) rope unit
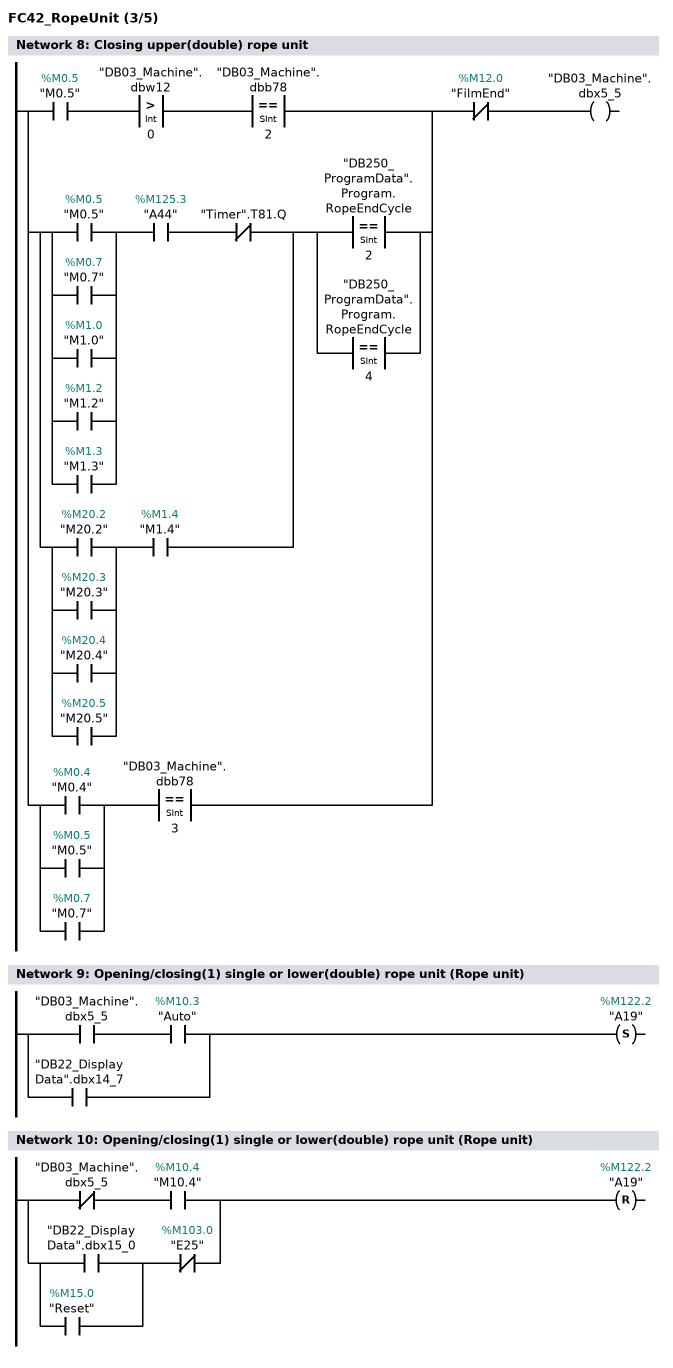
   RUNG wire#powerrail
      Contact( "M0.5" )
      { S7_Templates := "SrcType := Int" } GT_Contact(in1 := "DB03_Machine".dbw12, in2 := 0)
      { S7_Templates := "SrcType := SInt" } EQ_Contact(in1 := "DB03_Machine".dbb78, in2 := 2)
      wire#w1
      I_Contact( "FilmEnd" )
      Coil( "DB03_Machine".dbx5_5 )
   END_RUNG
   RUNG wire#powerrail
      Contact( "M0.5" )
      wire#w2
      Contact( "A44" )
      I_Contact( "Timer".T81.Q )
      wire#w3
      { S7_Templates := "SrcType := SInt" } EQ_Contact(in1 := "DB250_ProgramData".Program.RopeEndCycle, in2 := 2)
   END_RUNG wire#w1
   RUNG wire#powerrail
      Contact( "M0.7" )
   END_RUNG wire#w2
   RUNG wire#powerrail
      Contact( "M1.0" )
   END_RUNG wire#w2
   RUNG wire#powerrail
      Contact( "M1.2" )
   END_RUNG wire#w2
   RUNG wire#powerrail
      Contact( "M1.3" )
   END_RUNG wire#w2
   RUNG wire#powerrail
      Contact( "M20.2" )
      wire#w4
      Contact( "M1.4" )
   END_RUNG wire#w3
   RUNG wire#powerrail
      Contact( "M20.3" )
   END_RUNG wire#w4
   RUNG wire#powerrail
      Contact( "M20.4" )
   END_RUNG wire#w4
   RUNG wire#powerrail
      Contact( "M20.5" )
   END_RUNG wire#w4
   RUNG wire#w3
      { S7_Templates := "SrcType := SInt" } EQ_Contact(in1 := "DB250_ProgramData".Program.RopeEndCycle, in2 := 4)
   END_RUNG wire#w1
   RUNG wire#powerrail
      Contact( "M0.4" )
      wire#w5
      { S7_Templates := "SrcType := SInt" } EQ_Contact(in1 := "DB03_Machine".dbb78, in2 := 3)
   END_RUNG wire#w1
   RUNG wire#powerrail
      Contact( "M0.5" )
   END_RUNG wire#w5
   RUNG wire#powerrail
      Contact( "M0.7" )
   END_RUNG wire#w5
   // the same network as SCL:
   "DB03_Machine".dbx5_5 := (("M0.5" AND ("DB03_Machine".dbw12 > 0) AND ("DB03_Machine".dbb78 = 2)) OR (((("M0.5" OR "M0.7" OR "M1.0" OR "M1.2" OR "M1.3") AND "A44" AND NOT "Timer".T81.Q) OR (("M20.2" OR "M20.3" OR "M20.4" OR "M20.5") AND "M1.4")) AND (("DB250_ProgramData".Program.RopeEndCycle = 2) OR ("DB250_ProgramData".Program.RopeEndCycle = 4))) OR (("M0.4" OR "M0.5" OR "M0.7") AND ("DB03_Machine".dbb78 = 3))) AND NOT "FilmEnd";
END_REGION

REGION Network 9: Opening/closing(1) single or lower(double) rope unit (Rope unit)
   RUNG wire#powerrail
      Contact( "DB03_Machine".dbx5_5 )
      Contact( "Auto" )
      wire#w1
      S_Coil( "A19" )
   END_RUNG
   RUNG wire#powerrail
      Contact( "DB22_DisplayData".dbx14_7 )
   END_RUNG wire#w1
   // the same network as SCL:
   IF ("DB03_Machine".dbx5_5 AND "Auto") OR "DB22_DisplayData".dbx14_7 THEN "A19" := TRUE; END_IF;
END_REGION

REGION Network 10: Opening/closing(1) single or lower(double) rope unit (Rope unit)
   RUNG wire#powerrail
      I_Contact( "DB03_Machine".dbx5_5 )
      Contact( "M10.4" )
      wire#w1
      R_Coil( "A19" )
   END_RUNG
   RUNG wire#powerrail
      Contact( "DB22_DisplayData".dbx15_0 )
      wire#w2
      I_Contact( "E25" )
   END_RUNG wire#w1
   RUNG wire#powerrail
      Contact( "Reset" )
   END_RUNG wire#w2
   // the same network as SCL:
   IF (NOT "DB03_Machine".dbx5_5 AND "M10.4") OR (("DB22_DisplayData".dbx15_0 OR "Reset") AND NOT "E25") THEN
       "A19" := FALSE;
   END_IF;
END_REGION

REGION Network 11: Alarm 27: Timeout for rope unit open/close (Rope unit)
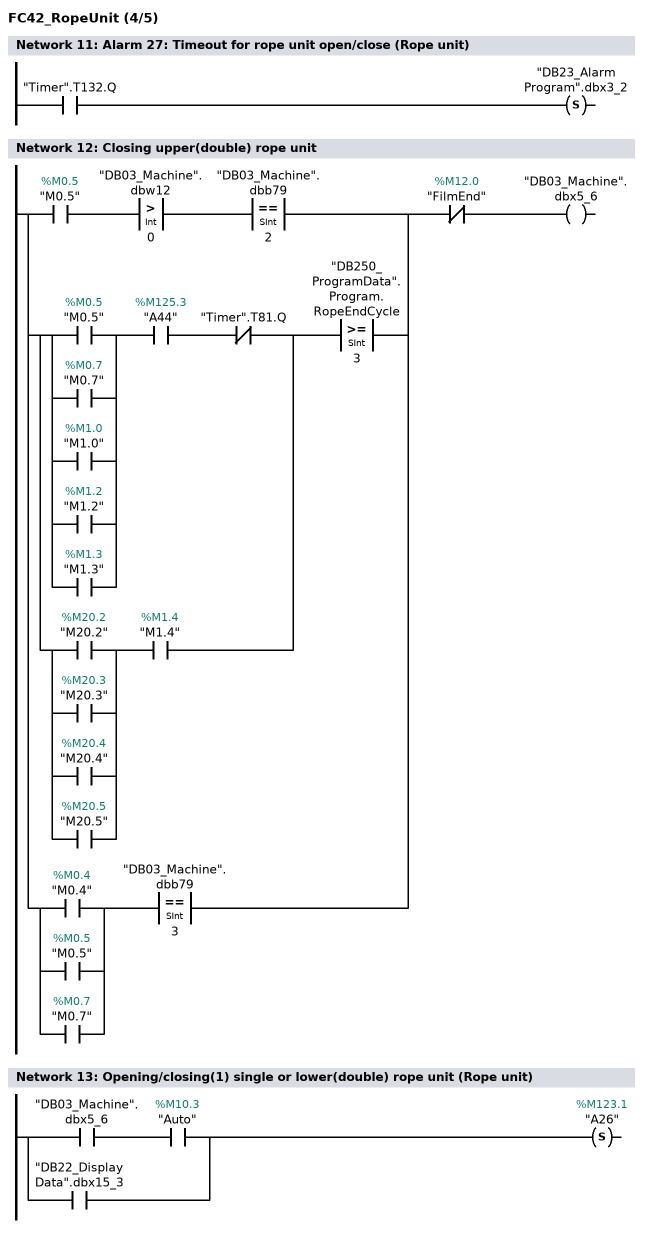
   RUNG wire#powerrail
      Contact( "Timer".T132.Q )
      S_Coil( "DB23_AlarmProgram".dbx3_2 )
   END_RUNG
   // the same network as SCL:
   IF "Timer".T132.Q THEN "DB23_AlarmProgram".dbx3_2 := TRUE; END_IF;
END_REGION

REGION Network 12: Closing upper(double) rope unit
   RUNG wire#powerrail
      Contact( "M0.5" )
      { S7_Templates := "SrcType := Int" } GT_Contact(in1 := "DB03_Machine".dbw12, in2 := 0)
      { S7_Templates := "SrcType := SInt" } EQ_Contact(in1 := "DB03_Machine".dbb79, in2 := 2)
      wire#w1
      I_Contact( "FilmEnd" )
      Coil( "DB03_Machine".dbx5_6 )
   END_RUNG
   RUNG wire#powerrail
      Contact( "M0.5" )
      wire#w2
      Contact( "A44" )
      I_Contact( "Timer".T81.Q )
      wire#w3
      { S7_Templates := "SrcType := SInt" } GE_Contact(in1 := "DB250_ProgramData".Program.RopeEndCycle, in2 := 3)
   END_RUNG wire#w1
   RUNG wire#powerrail
      Contact( "M0.7" )
   END_RUNG wire#w2
   RUNG wire#powerrail
      Contact( "M1.0" )
   END_RUNG wire#w2
   RUNG wire#powerrail
      Contact( "M1.2" )
   END_RUNG wire#w2
   RUNG wire#powerrail
      Contact( "M1.3" )
   END_RUNG wire#w2
   RUNG wire#powerrail
      Contact( "M20.2" )
      wire#w4
      Contact( "M1.4" )
   END_RUNG wire#w3
   RUNG wire#powerrail
      Contact( "M20.3" )
   END_RUNG wire#w4
   RUNG wire#powerrail
      Contact( "M20.4" )
   END_RUNG wire#w4
   RUNG wire#powerrail
      Contact( "M20.5" )
   END_RUNG wire#w4
   RUNG wire#powerrail
      Contact( "M0.4" )
      wire#w5
      { S7_Templates := "SrcType := SInt" } EQ_Contact(in1 := "DB03_Machine".dbb79, in2 := 3)
   END_RUNG wire#w1
   RUNG wire#powerrail
      Contact( "M0.5" )
   END_RUNG wire#w5
   RUNG wire#powerrail
      Contact( "M0.7" )
   END_RUNG wire#w5
   // the same network as SCL:
   "DB03_Machine".dbx5_6 := (("M0.5" AND ("DB03_Machine".dbw12 > 0) AND ("DB03_Machine".dbb79 = 2)) OR (((("M0.5" OR "M0.7" OR "M1.0" OR "M1.2" OR "M1.3") AND "A44" AND NOT "Timer".T81.Q) OR (("M20.2" OR "M20.3" OR "M20.4" OR "M20.5") AND "M1.4")) AND ("DB250_ProgramData".Program.RopeEndCycle >= 3)) OR (("M0.4" OR "M0.5" OR "M0.7") AND ("DB03_Machine".dbb79 = 3))) AND NOT "FilmEnd";
END_REGION

REGION Network 13: Opening/closing(1) single or lower(double) rope unit (Rope unit)
   RUNG wire#powerrail
      Contact( "DB03_Machine".dbx5_6 )
      Contact( "Auto" )
      wire#w1
      S_Coil( "A26" )
   END_RUNG
   RUNG wire#powerrail
      Contact( "DB22_DisplayData".dbx15_3 )
   END_RUNG wire#w1
   // the same network as SCL:
   IF ("DB03_Machine".dbx5_6 AND "Auto") OR "DB22_DisplayData".dbx15_3 THEN "A26" := TRUE; END_IF;
END_REGION

REGION Network 14: Opening/closing(1) single or lower(double) rope unit (Rope unit)
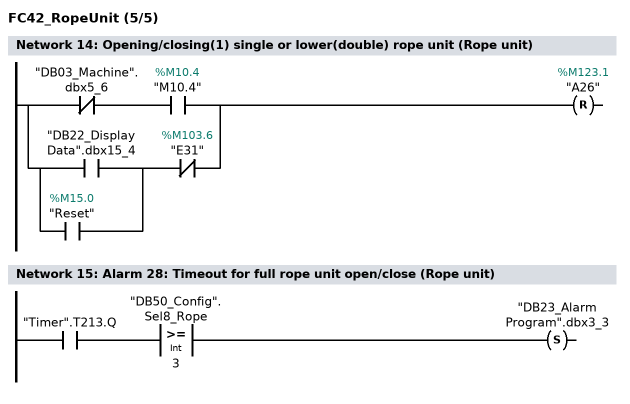
   RUNG wire#powerrail
      I_Contact( "DB03_Machine".dbx5_6 )
      Contact( "M10.4" )
      wire#w1
      R_Coil( "A26" )
   END_RUNG
   RUNG wire#powerrail
      Contact( "DB22_DisplayData".dbx15_4 )
      wire#w2
      I_Contact( "E31" )
   END_RUNG wire#w1
   RUNG wire#powerrail
      Contact( "Reset" )
   END_RUNG wire#w2
   // the same network as SCL:
   IF (NOT "DB03_Machine".dbx5_6 AND "M10.4") OR (("DB22_DisplayData".dbx15_4 OR "Reset") AND NOT "E31") THEN
       "A26" := FALSE;
   END_IF;
END_REGION

REGION Network 15: Alarm 28: Timeout for full rope unit open/close (Rope unit)
   RUNG wire#powerrail
      Contact( "Timer".T213.Q )
      { S7_Templates := "SrcType := Int" } GE_Contact(in1 := "DB50_Config".Sel8_Rope, in2 := 3)
      S_Coil( "DB23_AlarmProgram".dbx3_3 )
   END_RUNG
   // the same network as SCL:
   IF "Timer".T213.Q AND ("DB50_Config".Sel8_Rope >= 3) THEN "DB23_AlarmProgram".dbx3_3 := TRUE; END_IF;
END_REGION
END_FUNCTION

FUNCTION "FC05_TechnoplatOutput" : Void   // FC5, LAD
TITLE = Machine output
{ S7_Optimized_Access := 'FALSE' }
AUTHOR : Robopac
VERSION : 0.0
// stored: AutoNumber false, IsIECCheckEnabled false, SetENOAutomatically false, UDAEnableTagReadback false
   VAR_INPUT
      PHASE : Bool;
      FASTSPEED : Bool;
   END_VAR
   VAR_TEMP
      SuppSpeed : Bool;
      wTemp : Int;
      DwTemp : DInt;
      wTemp2 : Int;
      wTemp3 : Int;
      U201_START : Bool;
      U201_DIR : Bool;
      U201_SP : Int;
      U221_START : Bool;
      U221_DIR : Bool;
      U221_SP : Int;
      DwTemp2 : DInt;
   END_VAR
   VAR_TEMP   // added for the SCL form of the ladder/FBD networks
      _w1 : Bool;
   END_VAR
BEGIN

REGION Network 1: Emergency mode lamp (Helix)
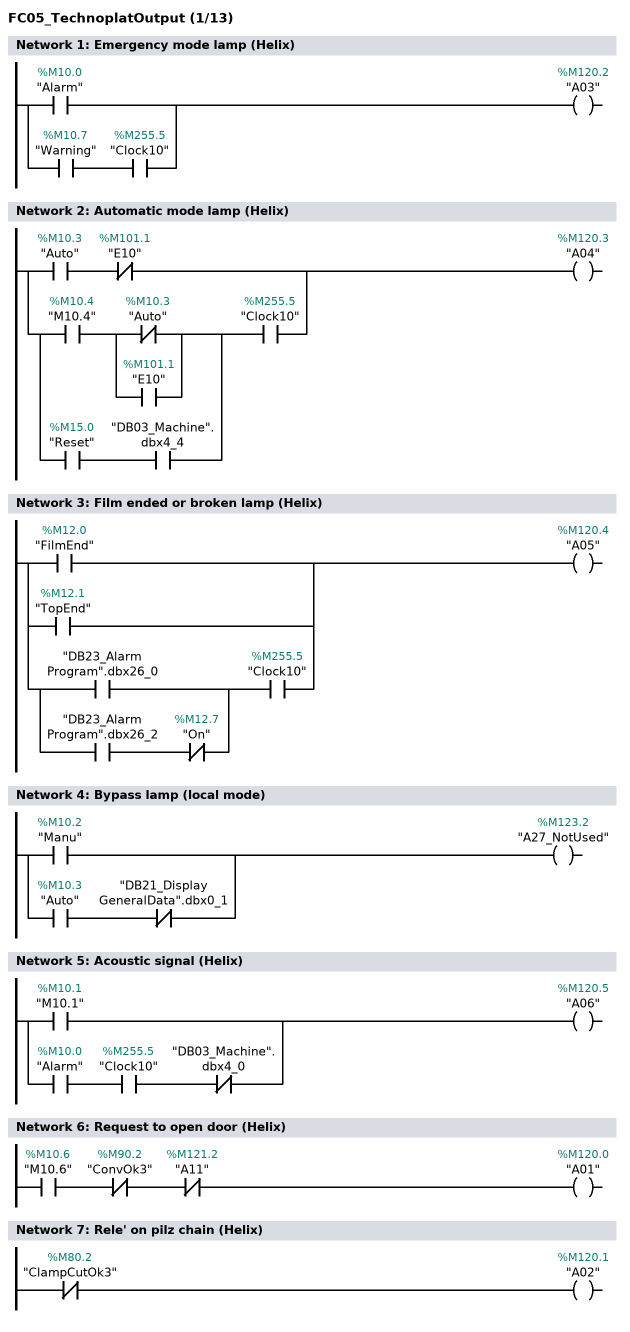
   RUNG wire#powerrail
      Contact( "Alarm" )
      wire#w1
      Coil( "A03" )
   END_RUNG
   RUNG wire#powerrail
      Contact( "Warning" )
      Contact( "Clock10" )
   END_RUNG wire#w1
   // the same network as SCL:
   "A03" := "Alarm" OR ("Warning" AND "Clock10");
END_REGION

REGION Network 2: Automatic mode lamp (Helix)
   RUNG wire#powerrail
      Contact( "Auto" )
      I_Contact( "E10" )
      wire#w1
      Coil( "A04" )
   END_RUNG
   RUNG wire#powerrail
      Contact( "M10.4" )
      wire#w2
      I_Contact( "Auto" )
      wire#w3
      Contact( "Clock10" )
   END_RUNG wire#w1
   RUNG wire#w2
      Contact( "E10" )
   END_RUNG wire#w3
   RUNG wire#powerrail
      Contact( "Reset" )
      Contact( "DB03_Machine".dbx4_4 )
   END_RUNG wire#w3
   // the same network as SCL:
   "A04" := ("Auto" AND NOT "E10") OR ((("M10.4" AND (NOT "Auto" OR "E10")) OR ("Reset" AND "DB03_Machine".dbx4_4)) AND "Clock10");
END_REGION

REGION Network 3: Film ended or broken lamp (Helix)
   RUNG wire#powerrail
      Contact( "FilmEnd" )
      wire#w1
      Coil( "A05" )
   END_RUNG
   RUNG wire#powerrail
      Contact( "TopEnd" )
   END_RUNG wire#w1
   RUNG wire#powerrail
      Contact( "DB23_AlarmProgram".dbx26_0 )
      wire#w2
      Contact( "Clock10" )
   END_RUNG wire#w1
   RUNG wire#powerrail
      Contact( "DB23_AlarmProgram".dbx26_2 )
      I_Contact( "On" )
   END_RUNG wire#w2
   // the same network as SCL:
   "A05" := "FilmEnd" OR "TopEnd" OR (("DB23_AlarmProgram".dbx26_0 OR ("DB23_AlarmProgram".dbx26_2 AND NOT "On")) AND "Clock10");
END_REGION

REGION Network 4: Bypass lamp (local mode)
   RUNG wire#powerrail
      Contact( "Manu" )
      wire#w1
      Coil( "A27_NotUsed" )
   END_RUNG
   RUNG wire#powerrail
      Contact( "Auto" )
      I_Contact( "DB21_DisplayGeneralData".dbx0_1 )
   END_RUNG wire#w1
   // the same network as SCL:
   "A27_NotUsed" := "Manu" OR ("Auto" AND NOT "DB21_DisplayGeneralData".dbx0_1);
END_REGION

REGION Network 5: Acoustic signal (Helix)
   RUNG wire#powerrail
      Contact( "M10.1" )
      wire#w1
      Coil( "A06" )
   END_RUNG
   RUNG wire#powerrail
      Contact( "Alarm" )
      Contact( "Clock10" )
      I_Contact( "DB03_Machine".dbx4_0 )
   END_RUNG wire#w1
   // the same network as SCL:
   "A06" := "M10.1" OR ("Alarm" AND "Clock10" AND NOT "DB03_Machine".dbx4_0);
END_REGION

REGION Network 6: Request to open door (Helix)
   RUNG wire#powerrail
      Contact( "M10.6" )
      I_Contact( "ConvOk3" )
      I_Contact( "A11" )
      Coil( "A01" )
   END_RUNG
   // the same network as SCL:
   "A01" := "M10.6" AND NOT "ConvOk3" AND NOT "A11";
END_REGION

REGION Network 7: Rele' on pilz chain (Helix)
   RUNG wire#powerrail
      I_Contact( "ClampCutOk3" )
      Coil( "A02" )
   END_RUNG
   // the same network as SCL:
   "A02" := NOT "ClampCutOk3";
END_REGION

REGION Network 8: Table rotation forward
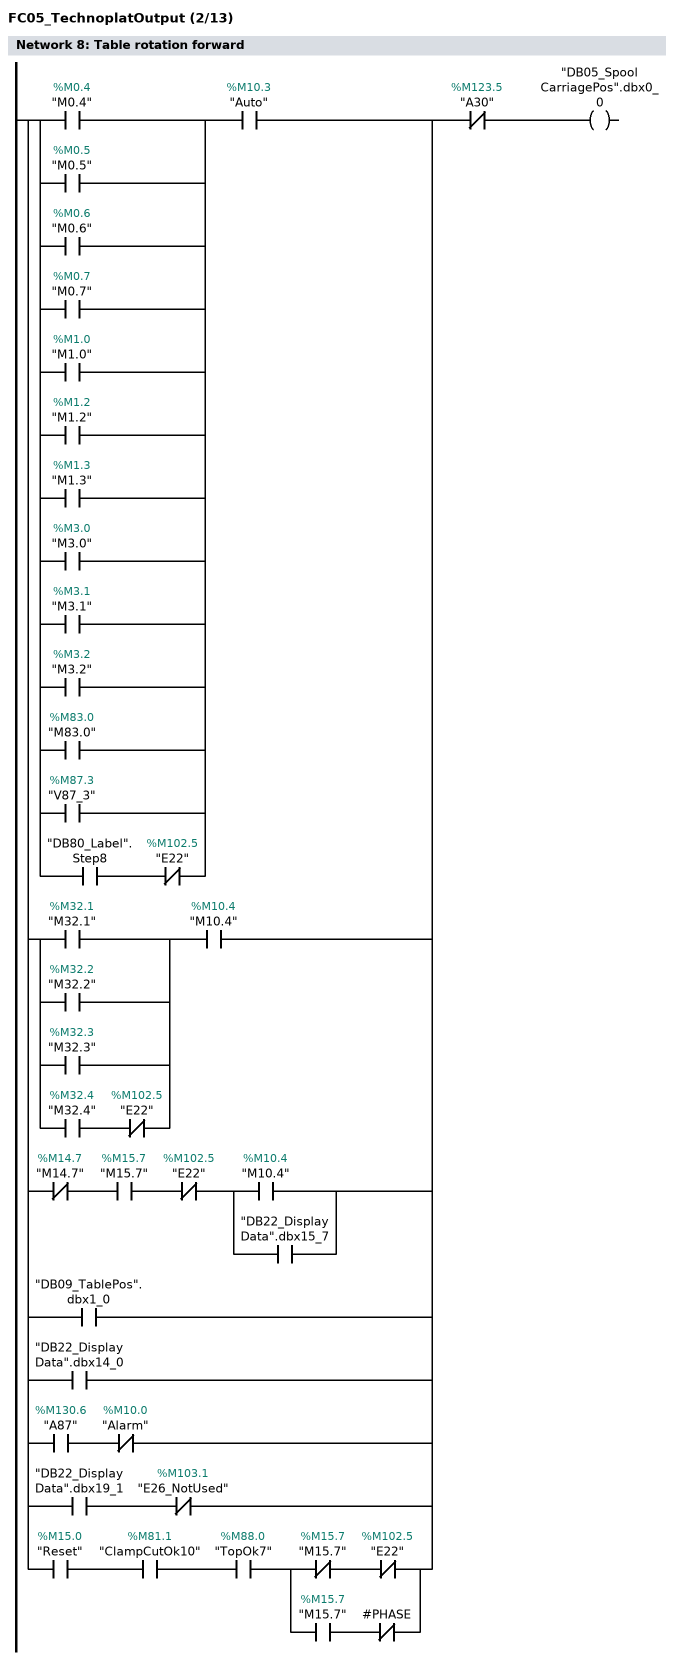
   RUNG wire#powerrail
      Contact( "M0.4" )
      wire#w1
      Contact( "Auto" )
      wire#w2
      I_Contact( "A30" )
      Coil( "DB05_SpoolCarriagePos".dbx0_0 )
   END_RUNG
   RUNG wire#powerrail
      Contact( "M0.5" )
   END_RUNG wire#w1
   RUNG wire#powerrail
      Contact( "M0.6" )
   END_RUNG wire#w1
   RUNG wire#powerrail
      Contact( "M0.7" )
   END_RUNG wire#w1
   RUNG wire#powerrail
      Contact( "M1.0" )
   END_RUNG wire#w1
   RUNG wire#powerrail
      Contact( "M1.2" )
   END_RUNG wire#w1
   RUNG wire#powerrail
      Contact( "M1.3" )
   END_RUNG wire#w1
   RUNG wire#powerrail
      Contact( "M3.0" )
   END_RUNG wire#w1
   RUNG wire#powerrail
      Contact( "M3.1" )
   END_RUNG wire#w1
   RUNG wire#powerrail
      Contact( "M3.2" )
   END_RUNG wire#w1
   RUNG wire#powerrail
      Contact( "M83.0" )
   END_RUNG wire#w1
   RUNG wire#powerrail
      Contact( "V87_3" )
   END_RUNG wire#w1
   RUNG wire#powerrail
      Contact( "DB80_Label".Step8 )
      I_Contact( "E22" )
   END_RUNG wire#w1
   RUNG wire#powerrail
      Contact( "M32.1" )
      wire#w3
      Contact( "M10.4" )
   END_RUNG wire#w2
   RUNG wire#powerrail
      Contact( "M32.2" )
   END_RUNG wire#w3
   RUNG wire#powerrail
      Contact( "M32.3" )
   END_RUNG wire#w3
   RUNG wire#powerrail
      Contact( "M32.4" )
      I_Contact( "E22" )
   END_RUNG wire#w3
   RUNG wire#powerrail
      I_Contact( "M14.7" )
      Contact( "M15.7" )
      I_Contact( "E22" )
      wire#w4
      Contact( "M10.4" )
   END_RUNG wire#w2
   RUNG wire#w4
      Contact( "DB22_DisplayData".dbx15_7 )
   END_RUNG wire#w2
   RUNG wire#powerrail
      Contact( "DB09_TablePos".dbx1_0 )
   END_RUNG wire#w2
   RUNG wire#powerrail
      Contact( "DB22_DisplayData".dbx14_0 )
   END_RUNG wire#w2
   RUNG wire#powerrail
      Contact( "A87" )
      I_Contact( "Alarm" )
   END_RUNG wire#w2
   RUNG wire#powerrail
      Contact( "DB22_DisplayData".dbx19_1 )
      I_Contact( "E26_NotUsed" )
   END_RUNG wire#w2
   RUNG wire#powerrail
      Contact( "Reset" )
      Contact( "ClampCutOk10" )
      Contact( "TopOk7" )
      wire#w5
      I_Contact( "M15.7" )
      I_Contact( "E22" )
   END_RUNG wire#w2
   RUNG wire#w5
      Contact( "M15.7" )
      I_Contact( #PHASE )
   END_RUNG wire#w2
   // the same network as SCL:
   "DB05_SpoolCarriagePos".dbx0_0 := ((("M0.4" OR "M0.5" OR "M0.6" OR "M0.7" OR "M1.0" OR "M1.2" OR "M1.3" OR "M3.0" OR "M3.1" OR "M3.2" OR "M83.0" OR "V87_3" OR ("DB80_Label".Step8 AND NOT "E22")) AND "Auto") OR (("M32.1" OR "M32.2" OR "M32.3" OR ("M32.4" AND NOT "E22")) AND "M10.4") OR (NOT "M14.7" AND "M15.7" AND NOT "E22" AND ("M10.4" OR "DB22_DisplayData".dbx15_7)) OR "DB09_TablePos".dbx1_0 OR "DB22_DisplayData".dbx14_0 OR ("A87" AND NOT "Alarm") OR ("DB22_DisplayData".dbx19_1 AND NOT "E26_NotUsed") OR ("Reset" AND "ClampCutOk10" AND "TopOk7" AND ((NOT "M15.7" AND NOT "E22") OR ("M15.7" AND NOT #PHASE)))) AND NOT "A30";
END_REGION

REGION Network 9: Table rotation backward
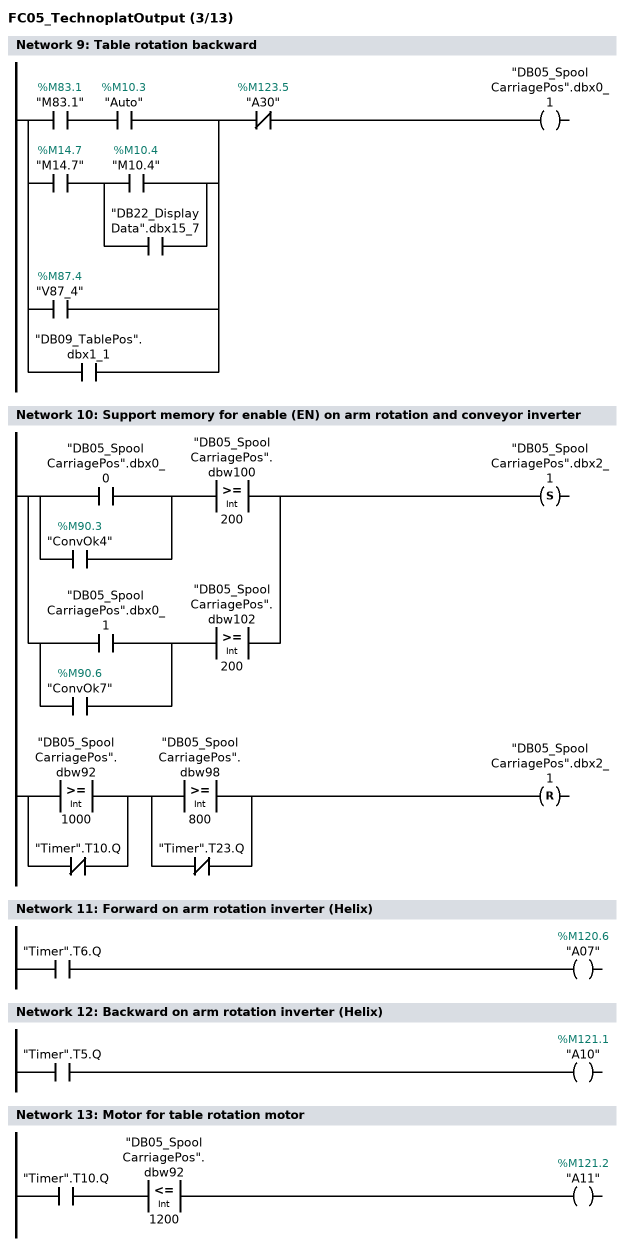
   RUNG wire#powerrail
      Contact( "M83.1" )
      Contact( "Auto" )
      wire#w1
      I_Contact( "A30" )
      Coil( "DB05_SpoolCarriagePos".dbx0_1 )
   END_RUNG
   RUNG wire#powerrail
      Contact( "M14.7" )
      wire#w2
      Contact( "M10.4" )
   END_RUNG wire#w1
   RUNG wire#w2
      Contact( "DB22_DisplayData".dbx15_7 )
   END_RUNG wire#w1
   RUNG wire#powerrail
      Contact( "V87_4" )
   END_RUNG wire#w1
   RUNG wire#powerrail
      Contact( "DB09_TablePos".dbx1_1 )
   END_RUNG wire#w1
   // the same network as SCL:
   "DB05_SpoolCarriagePos".dbx0_1 := (("M83.1" AND "Auto") OR ("M14.7" AND ("M10.4" OR "DB22_DisplayData".dbx15_7)) OR "V87_4" OR "DB09_TablePos".dbx1_1) AND NOT "A30";
END_REGION

REGION Network 10: Support memory for enable (EN) on arm rotation and conveyor inverter
   RUNG wire#powerrail
      Contact( "DB05_SpoolCarriagePos".dbx0_0 )
      wire#w1
      { S7_Templates := "SrcType := Int" } GE_Contact(in1 := "DB05_SpoolCarriagePos".dbw100, in2 := 200)
      wire#w2
      S_Coil( "DB05_SpoolCarriagePos".dbx2_1 )
   END_RUNG
   RUNG wire#powerrail
      Contact( "ConvOk4" )
   END_RUNG wire#w1
   RUNG wire#powerrail
      Contact( "DB05_SpoolCarriagePos".dbx0_1 )
      wire#w3
      { S7_Templates := "SrcType := Int" } GE_Contact(in1 := "DB05_SpoolCarriagePos".dbw102, in2 := 200)
   END_RUNG wire#w2
   RUNG wire#powerrail
      Contact( "ConvOk7" )
   END_RUNG wire#w3
   RUNG wire#powerrail
      { S7_Templates := "SrcType := Int" } GE_Contact(in1 := "DB05_SpoolCarriagePos".dbw92, in2 := 1000)
      wire#w4
      { S7_Templates := "SrcType := Int" } GE_Contact(in1 := "DB05_SpoolCarriagePos".dbw98, in2 := 800)
      wire#w5
      R_Coil( "DB05_SpoolCarriagePos".dbx2_1 )
   END_RUNG
   RUNG wire#powerrail
      I_Contact( "Timer".T10.Q )
   END_RUNG wire#w4
   RUNG wire#w4
      I_Contact( "Timer".T23.Q )
   END_RUNG wire#w5
   // the same network as SCL:
   IF (("DB05_SpoolCarriagePos".dbx0_0 OR "ConvOk4") AND ("DB05_SpoolCarriagePos".dbw100 >= 200)) OR (("DB05_SpoolCarriagePos".dbx0_1 OR "ConvOk7") AND ("DB05_SpoolCarriagePos".dbw102 >= 200)) THEN
       "DB05_SpoolCarriagePos".dbx2_1 := TRUE;
   END_IF;
   IF (("DB05_SpoolCarriagePos".dbw92 >= 1000) OR NOT "Timer".T10.Q) AND (("DB05_SpoolCarriagePos".dbw98 >= 800) OR NOT "Timer".T23.Q) THEN
       "DB05_SpoolCarriagePos".dbx2_1 := FALSE;
   END_IF;
END_REGION

REGION Network 11: Forward on arm rotation inverter (Helix)
   RUNG wire#powerrail
      Contact( "Timer".T6.Q )
      Coil( "A07" )
   END_RUNG
   // the same network as SCL:
   "A07" := "Timer".T6.Q;
END_REGION

REGION Network 12: Backward on arm rotation inverter (Helix)
   RUNG wire#powerrail
      Contact( "Timer".T5.Q )
      Coil( "A10" )
   END_RUNG
   // the same network as SCL:
   "A10" := "Timer".T5.Q;
END_REGION

REGION Network 13: Motor for table rotation motor
   RUNG wire#powerrail
      Contact( "Timer".T10.Q )
      { S7_Templates := "SrcType := Int" } LE_Contact(in1 := "DB05_SpoolCarriagePos".dbw92, in2 := 1200)
      Coil( "A11" )
   END_RUNG
   // the same network as SCL:
   "A11" := "Timer".T10.Q AND ("DB05_SpoolCarriagePos".dbw92 <= 1200);
END_REGION

REGION Network 14: Brake for table rotation motor (Technoplat)
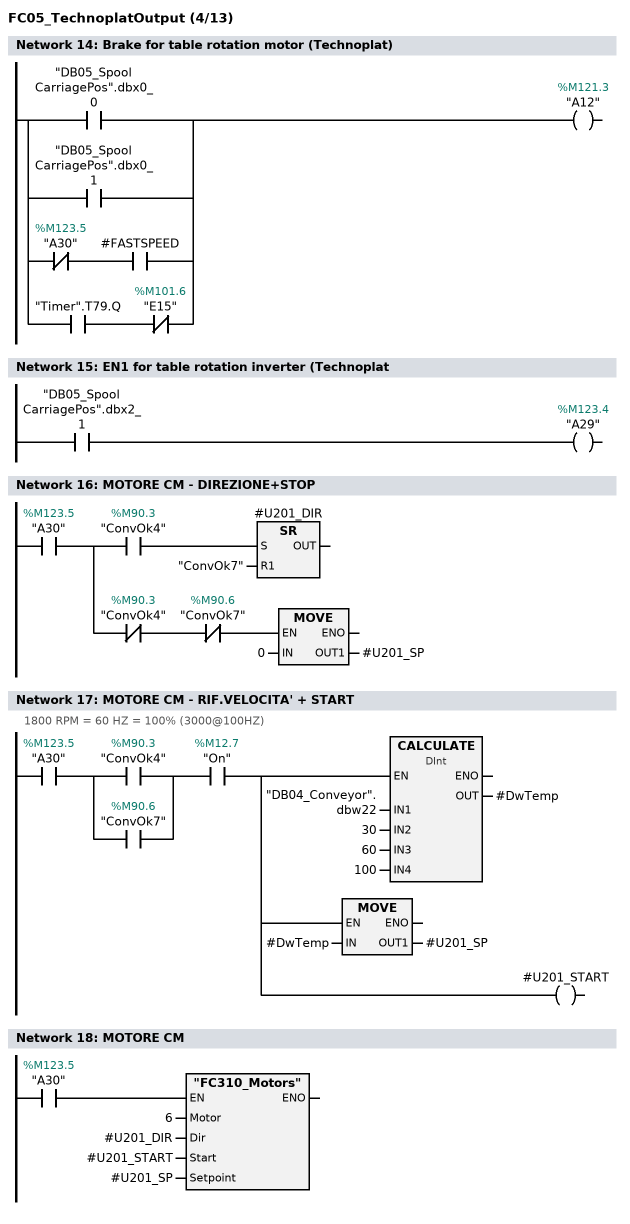
   RUNG wire#powerrail
      Contact( "DB05_SpoolCarriagePos".dbx0_0 )
      wire#w1
      Coil( "A12" )
   END_RUNG
   RUNG wire#powerrail
      Contact( "DB05_SpoolCarriagePos".dbx0_1 )
   END_RUNG wire#w1
   RUNG wire#powerrail
      I_Contact( "A30" )
      Contact( #FASTSPEED )
   END_RUNG wire#w1
   RUNG wire#powerrail
      Contact( "Timer".T79.Q )
      I_Contact( "E15" )
   END_RUNG wire#w1
   // the same network as SCL:
   "A12" := "DB05_SpoolCarriagePos".dbx0_0 OR "DB05_SpoolCarriagePos".dbx0_1 OR (NOT "A30" AND #FASTSPEED) OR ("Timer".T79.Q AND NOT "E15");
END_REGION

REGION Network 15: EN1 for table rotation inverter (Technoplat
   RUNG wire#powerrail
      Contact( "DB05_SpoolCarriagePos".dbx2_1 )
      Coil( "A29" )
   END_RUNG
   // the same network as SCL:
   "A29" := "DB05_SpoolCarriagePos".dbx2_1;
END_REGION

REGION Network 16: MOTORE CM - DIREZIONE+STOP
   RUNG wire#powerrail
      Contact( "A30" )
      wire#w1
      Contact( "ConvOk4" )
      S_SR(operand := #U201_DIR, r1 := "ConvOk7")
   END_RUNG
   RUNG wire#w1
      I_Contact( "ConvOk4" )
      I_Contact( "ConvOk7" )
      Move(in := 0, out1 => #U201_SP)
   END_RUNG
   // the same network as SCL:
   IF "A30" AND "ConvOk4" THEN
       #U201_DIR := TRUE;   // SR flip-flop
   END_IF;
   IF "ConvOk7" THEN #U201_DIR := FALSE; END_IF;
   IF "A30" AND NOT "ConvOk4" AND NOT "ConvOk7" THEN #U201_SP := 0; END_IF;
END_REGION

REGION Network 17: MOTORE CM - RIF.VELOCITA' + START
   // 1800 RPM = 60 HZ = 100% (3000@100HZ)
   RUNG wire#powerrail
      Contact( "A30" )
      wire#w1
      Contact( "ConvOk4" )
      wire#w2
      Contact( "On" )
      wire#w3
      { S7_Templates := "SrcType := DInt"; S7_Expression := "(IN1*IN2*IN3)/IN4" } Calculate(in1 := "DB04_Conveyor".dbw22, in2 := 30, in3 := 60, in4 := 100, out => #DwTemp)
   END_RUNG
   RUNG wire#w1
      Contact( "ConvOk7" )
   END_RUNG wire#w2
   RUNG wire#w3
      Move(in := #DwTemp, out1 => #U201_SP)
   END_RUNG
   RUNG wire#w3
      Coil( #U201_START )
   END_RUNG
   // the same network as SCL:
   #_w1 := "A30" AND ("ConvOk4" OR "ConvOk7") AND "On";
   IF #_w1 THEN
       #DwTemp := ("DB04_Conveyor".dbw22*30*60)/100;
       #U201_SP := #DwTemp;
   END_IF;
   #U201_START := #_w1;
END_REGION

REGION Network 18: MOTORE CM
   RUNG wire#powerrail
      Contact( "A30" )
      "FC310_Motors"(Motor := 6, Dir := #U201_DIR, Start := #U201_START, Setpoint := #U201_SP)
   END_RUNG
   // the same network as SCL:
   IF "A30" THEN
       "FC310_Motors"(Motor := 6, Dir := #U201_DIR, Start := #U201_START, Setpoint := #U201_SP);
   END_IF;
END_REGION

REGION Network 19: Positioning command for OFF3 U201 (ON=normal functioning/OFF fast stop)
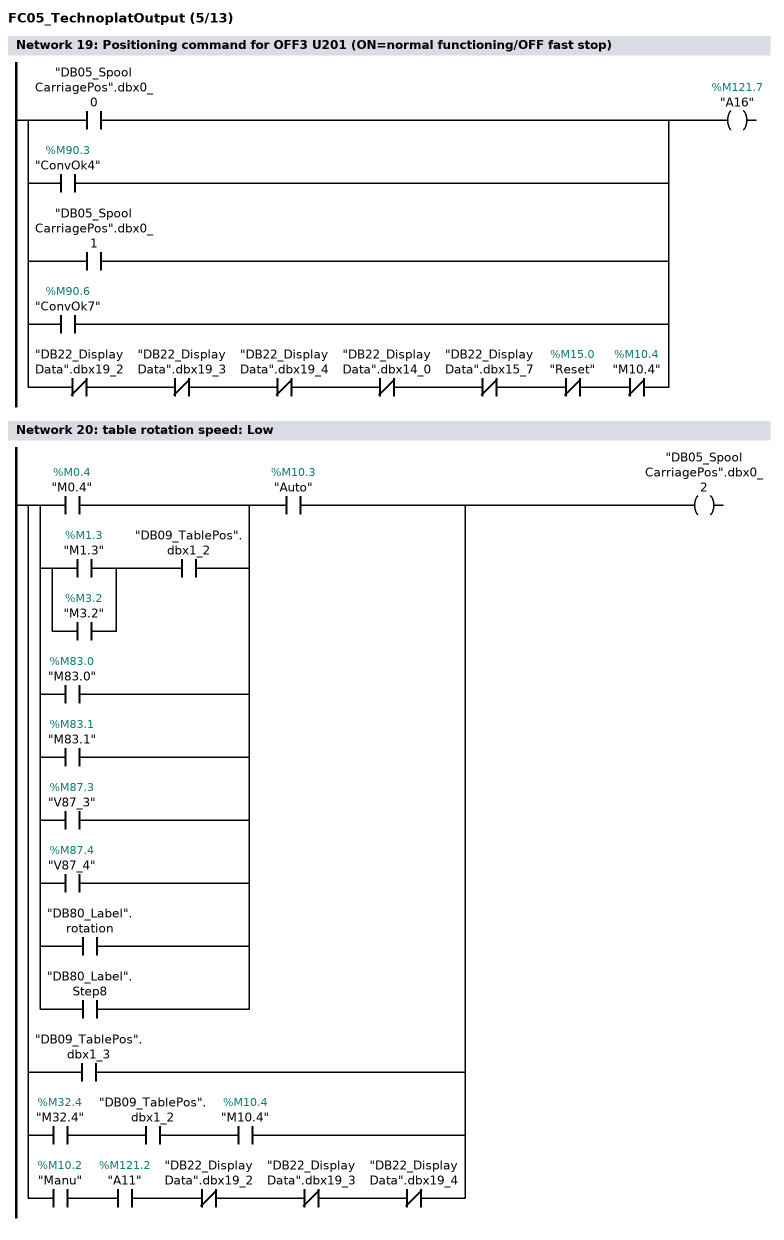
   RUNG wire#powerrail
      Contact( "DB05_SpoolCarriagePos".dbx0_0 )
      wire#w1
      Coil( "A16" )
   END_RUNG
   RUNG wire#powerrail
      Contact( "ConvOk4" )
   END_RUNG wire#w1
   RUNG wire#powerrail
      Contact( "DB05_SpoolCarriagePos".dbx0_1 )
   END_RUNG wire#w1
   RUNG wire#powerrail
      Contact( "ConvOk7" )
   END_RUNG wire#w1
   RUNG wire#powerrail
      I_Contact( "DB22_DisplayData".dbx19_2 )
      I_Contact( "DB22_DisplayData".dbx19_3 )
      I_Contact( "DB22_DisplayData".dbx19_4 )
      I_Contact( "DB22_DisplayData".dbx14_0 )
      I_Contact( "DB22_DisplayData".dbx15_7 )
      I_Contact( "Reset" )
      I_Contact( "M10.4" )
   END_RUNG wire#w1
   // the same network as SCL:
   "A16" := "DB05_SpoolCarriagePos".dbx0_0 OR "ConvOk4" OR "DB05_SpoolCarriagePos".dbx0_1 OR "ConvOk7" OR (NOT "DB22_DisplayData".dbx19_2 AND NOT "DB22_DisplayData".dbx19_3 AND NOT "DB22_DisplayData".dbx19_4 AND NOT "DB22_DisplayData".dbx14_0 AND NOT "DB22_DisplayData".dbx15_7 AND NOT "Reset" AND NOT "M10.4");
END_REGION

REGION Network 20: table rotation speed: Low
   RUNG wire#powerrail
      Contact( "M0.4" )
      wire#w1
      Contact( "Auto" )
      wire#w3
      Coil( "DB05_SpoolCarriagePos".dbx0_2 )
   END_RUNG
   RUNG wire#powerrail
      Contact( "M1.3" )
      wire#w2
      Contact( "DB09_TablePos".dbx1_2 )
   END_RUNG wire#w1
   RUNG wire#powerrail
      Contact( "M3.2" )
   END_RUNG wire#w2
   RUNG wire#powerrail
      Contact( "M83.0" )
   END_RUNG wire#w1
   RUNG wire#powerrail
      Contact( "M83.1" )
   END_RUNG wire#w1
   RUNG wire#powerrail
      Contact( "V87_3" )
   END_RUNG wire#w1
   RUNG wire#powerrail
      Contact( "V87_4" )
   END_RUNG wire#w1
   RUNG wire#powerrail
      Contact( "DB80_Label".rotation )
   END_RUNG wire#w1
   RUNG wire#powerrail
      Contact( "DB80_Label".Step8 )
   END_RUNG wire#w1
   RUNG wire#powerrail
      Contact( "DB09_TablePos".dbx1_3 )
   END_RUNG wire#w3
   RUNG wire#powerrail
      Contact( "M32.4" )
      Contact( "DB09_TablePos".dbx1_2 )
      Contact( "M10.4" )
   END_RUNG wire#w3
   RUNG wire#powerrail
      Contact( "Manu" )
      Contact( "A11" )
      I_Contact( "DB22_DisplayData".dbx19_2 )
      I_Contact( "DB22_DisplayData".dbx19_3 )
      I_Contact( "DB22_DisplayData".dbx19_4 )
   END_RUNG wire#w3
   // the same network as SCL:
   "DB05_SpoolCarriagePos".dbx0_2 := (("M0.4" OR (("M1.3" OR "M3.2") AND "DB09_TablePos".dbx1_2) OR "M83.0" OR "M83.1" OR "V87_3" OR "V87_4" OR "DB80_Label".rotation OR "DB80_Label".Step8) AND "Auto") OR "DB09_TablePos".dbx1_3 OR ("M32.4" AND "DB09_TablePos".dbx1_2 AND "M10.4") OR ("Manu" AND "A11" AND NOT "DB22_DisplayData".dbx19_2 AND NOT "DB22_DisplayData".dbx19_3 AND NOT "DB22_DisplayData".dbx19_4);
END_REGION

REGION Network 21: Table rotation speed: Middle 2 for welder contrast
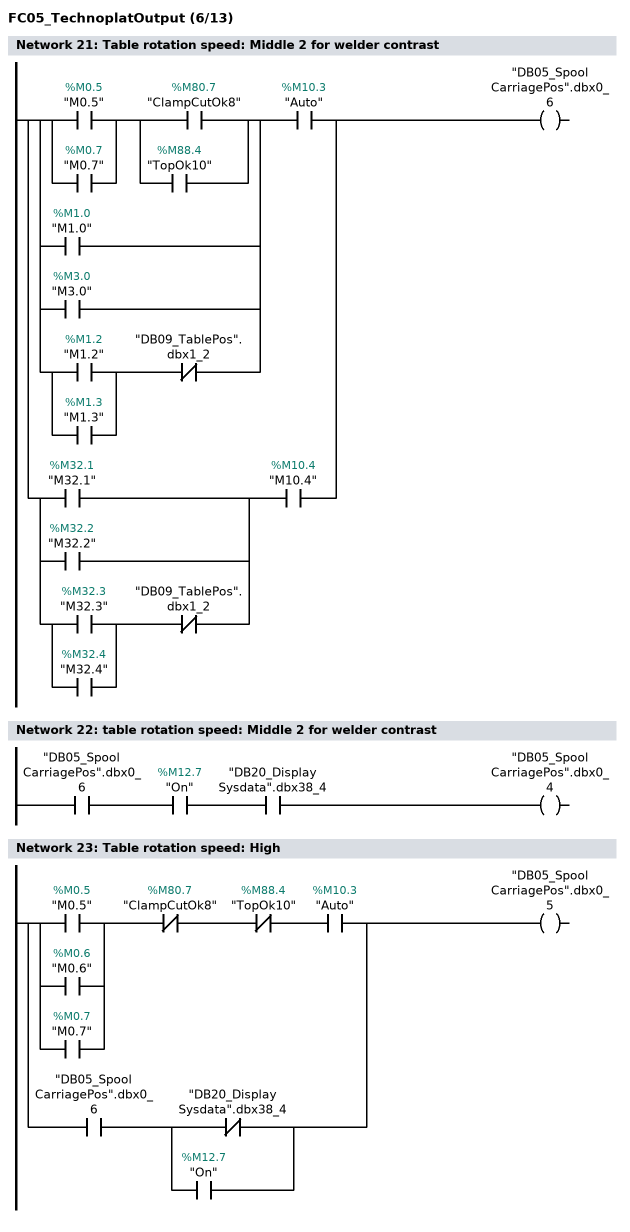
   RUNG wire#powerrail
      Contact( "M0.5" )
      wire#w1
      Contact( "ClampCutOk8" )
      wire#w2
      Contact( "Auto" )
      wire#w4
      Coil( "DB05_SpoolCarriagePos".dbx0_6 )
   END_RUNG
   RUNG wire#powerrail
      Contact( "M0.7" )
   END_RUNG wire#w1
   RUNG wire#w1
      Contact( "TopOk10" )
   END_RUNG wire#w2
   RUNG wire#powerrail
      Contact( "M1.0" )
   END_RUNG wire#w2
   RUNG wire#powerrail
      Contact( "M3.0" )
   END_RUNG wire#w2
   RUNG wire#powerrail
      Contact( "M1.2" )
      wire#w3
      I_Contact( "DB09_TablePos".dbx1_2 )
   END_RUNG wire#w2
   RUNG wire#powerrail
      Contact( "M1.3" )
   END_RUNG wire#w3
   RUNG wire#powerrail
      Contact( "M32.1" )
      wire#w5
      Contact( "M10.4" )
   END_RUNG wire#w4
   RUNG wire#powerrail
      Contact( "M32.2" )
   END_RUNG wire#w5
   RUNG wire#powerrail
      Contact( "M32.3" )
      wire#w6
      I_Contact( "DB09_TablePos".dbx1_2 )
   END_RUNG wire#w5
   RUNG wire#powerrail
      Contact( "M32.4" )
   END_RUNG wire#w6
   // the same network as SCL:
   "DB05_SpoolCarriagePos".dbx0_6 := (((("M0.5" OR "M0.7") AND ("ClampCutOk8" OR "TopOk10")) OR "M1.0" OR "M3.0" OR (("M1.2" OR "M1.3") AND NOT "DB09_TablePos".dbx1_2)) AND "Auto") OR (("M32.1" OR "M32.2" OR (("M32.3" OR "M32.4") AND NOT "DB09_TablePos".dbx1_2)) AND "M10.4");
END_REGION

REGION Network 22: table rotation speed: Middle 2 for welder contrast
   RUNG wire#powerrail
      Contact( "DB05_SpoolCarriagePos".dbx0_6 )
      Contact( "On" )
      Contact( "DB20_DisplaySysdata".dbx38_4 )
      Coil( "DB05_SpoolCarriagePos".dbx0_4 )
   END_RUNG
   // the same network as SCL:
   "DB05_SpoolCarriagePos".dbx0_4 := "DB05_SpoolCarriagePos".dbx0_6 AND "On" AND "DB20_DisplaySysdata".dbx38_4;
END_REGION

REGION Network 23: Table rotation speed: High
   RUNG wire#powerrail
      Contact( "M0.5" )
      wire#w1
      I_Contact( "ClampCutOk8" )
      I_Contact( "TopOk10" )
      Contact( "Auto" )
      wire#w2
      Coil( "DB05_SpoolCarriagePos".dbx0_5 )
   END_RUNG
   RUNG wire#powerrail
      Contact( "M0.6" )
   END_RUNG wire#w1
   RUNG wire#powerrail
      Contact( "M0.7" )
   END_RUNG wire#w1
   RUNG wire#powerrail
      Contact( "DB05_SpoolCarriagePos".dbx0_6 )
      wire#w3
      I_Contact( "DB20_DisplaySysdata".dbx38_4 )
   END_RUNG wire#w2
   RUNG wire#w3
      Contact( "On" )
   END_RUNG wire#w2
   // the same network as SCL:
   "DB05_SpoolCarriagePos".dbx0_5 := (("M0.5" OR "M0.6" OR "M0.7") AND NOT "ClampCutOk8" AND NOT "TopOk10" AND "Auto") OR ("DB05_SpoolCarriagePos".dbx0_6 AND (NOT "DB20_DisplaySysdata".dbx38_4 OR "On"));
END_REGION

REGION Network 24: Speed selection (X2-S4I) on arm rotation inverter (Technoplat)
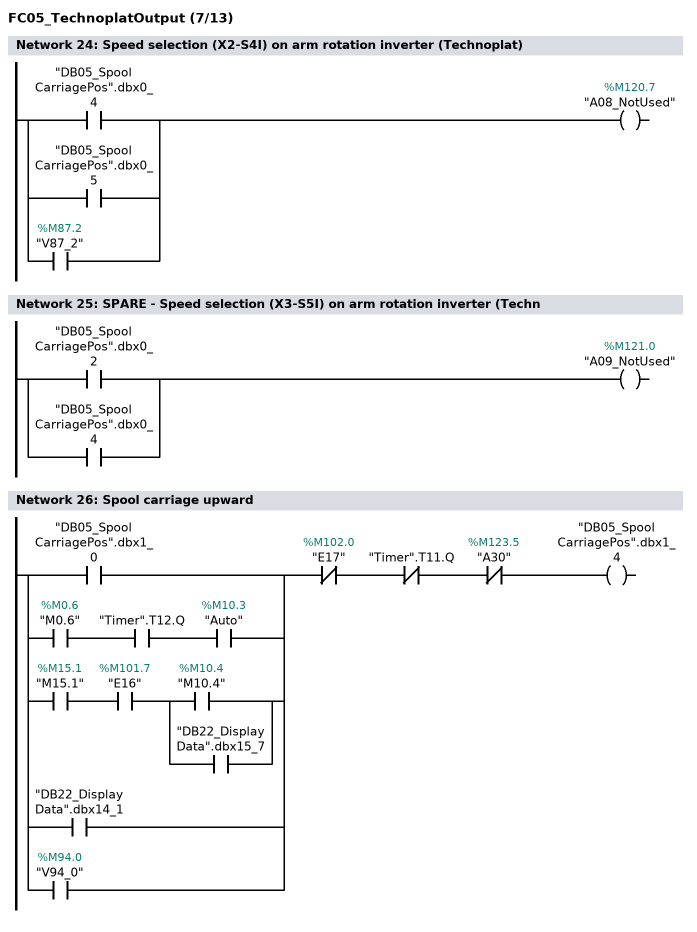
   RUNG wire#powerrail
      Contact( "DB05_SpoolCarriagePos".dbx0_4 )
      wire#w1
      Coil( "A08_NotUsed" )
   END_RUNG
   RUNG wire#powerrail
      Contact( "DB05_SpoolCarriagePos".dbx0_5 )
   END_RUNG wire#w1
   RUNG wire#powerrail
      Contact( "V87_2" )
   END_RUNG wire#w1
   // the same network as SCL:
   "A08_NotUsed" := "DB05_SpoolCarriagePos".dbx0_4 OR "DB05_SpoolCarriagePos".dbx0_5 OR "V87_2";
END_REGION

REGION Network 25: SPARE - Speed selection (X3-S5I) on arm rotation inverter (Techn
   RUNG wire#powerrail
      Contact( "DB05_SpoolCarriagePos".dbx0_2 )
      wire#w1
      Coil( "A09_NotUsed" )
   END_RUNG
   RUNG wire#powerrail
      Contact( "DB05_SpoolCarriagePos".dbx0_4 )
   END_RUNG wire#w1
   // the same network as SCL:
   "A09_NotUsed" := "DB05_SpoolCarriagePos".dbx0_2 OR "DB05_SpoolCarriagePos".dbx0_4;
END_REGION

REGION Network 26: Spool carriage upward
   RUNG wire#powerrail
      Contact( "DB05_SpoolCarriagePos".dbx1_0 )
      wire#w1
      I_Contact( "E17" )
      I_Contact( "Timer".T11.Q )
      I_Contact( "A30" )
      Coil( "DB05_SpoolCarriagePos".dbx1_4 )
   END_RUNG
   RUNG wire#powerrail
      Contact( "M0.6" )
      Contact( "Timer".T12.Q )
      Contact( "Auto" )
   END_RUNG wire#w1
   RUNG wire#powerrail
      Contact( "M15.1" )
      Contact( "E16" )
      wire#w2
      Contact( "M10.4" )
   END_RUNG wire#w1
   RUNG wire#w2
      Contact( "DB22_DisplayData".dbx15_7 )
   END_RUNG wire#w1
   RUNG wire#powerrail
      Contact( "DB22_DisplayData".dbx14_1 )
   END_RUNG wire#w1
   RUNG wire#powerrail
      Contact( "V94_0" )
   END_RUNG wire#w1
   // the same network as SCL:
   "DB05_SpoolCarriagePos".dbx1_4 := ("DB05_SpoolCarriagePos".dbx1_0 OR ("M0.6" AND "Timer".T12.Q AND "Auto") OR ("M15.1" AND "E16" AND ("M10.4" OR "DB22_DisplayData".dbx15_7)) OR "DB22_DisplayData".dbx14_1 OR "V94_0") AND NOT "E17" AND NOT "Timer".T11.Q AND NOT "A30";
END_REGION

REGION Network 27: Spool carriage downward
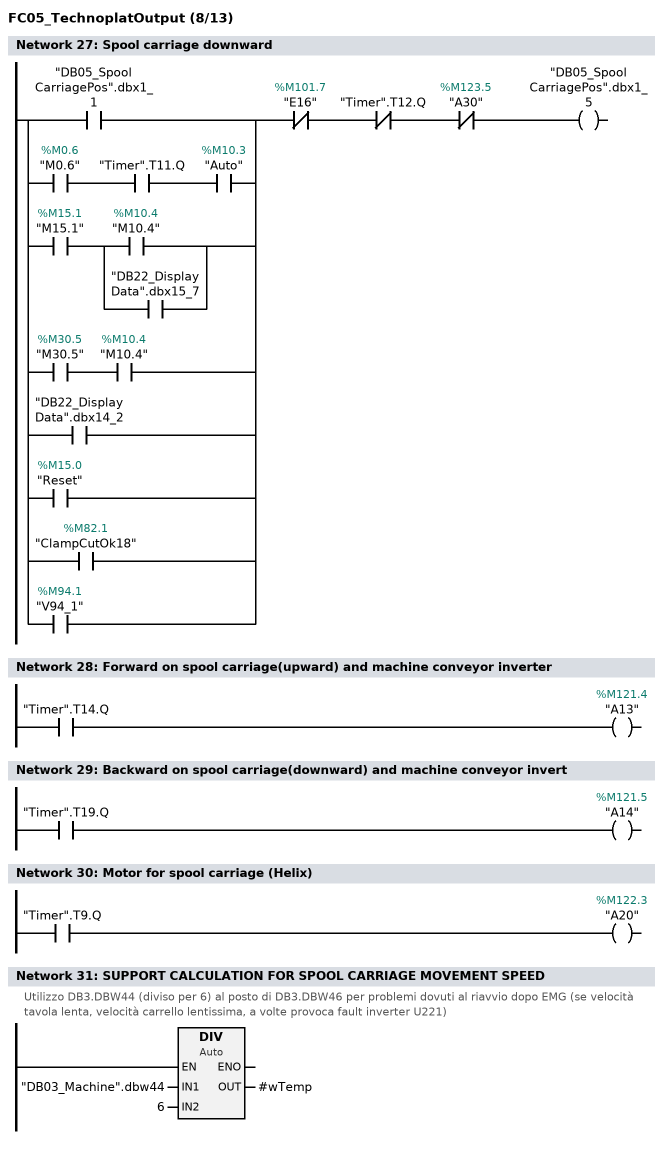
   RUNG wire#powerrail
      Contact( "DB05_SpoolCarriagePos".dbx1_1 )
      wire#w1
      I_Contact( "E16" )
      I_Contact( "Timer".T12.Q )
      I_Contact( "A30" )
      Coil( "DB05_SpoolCarriagePos".dbx1_5 )
   END_RUNG
   RUNG wire#powerrail
      Contact( "M0.6" )
      Contact( "Timer".T11.Q )
      Contact( "Auto" )
   END_RUNG wire#w1
   RUNG wire#powerrail
      Contact( "M15.1" )
      wire#w2
      Contact( "M10.4" )
   END_RUNG wire#w1
   RUNG wire#w2
      Contact( "DB22_DisplayData".dbx15_7 )
   END_RUNG wire#w1
   RUNG wire#powerrail
      Contact( "M30.5" )
      Contact( "M10.4" )
   END_RUNG wire#w1
   RUNG wire#powerrail
      Contact( "DB22_DisplayData".dbx14_2 )
   END_RUNG wire#w1
   RUNG wire#powerrail
      Contact( "Reset" )
   END_RUNG wire#w1
   RUNG wire#powerrail
      Contact( "ClampCutOk18" )
   END_RUNG wire#w1
   RUNG wire#powerrail
      Contact( "V94_1" )
   END_RUNG wire#w1
   // the same network as SCL:
   "DB05_SpoolCarriagePos".dbx1_5 := ("DB05_SpoolCarriagePos".dbx1_1 OR ("M0.6" AND "Timer".T11.Q AND "Auto") OR ("M15.1" AND ("M10.4" OR "DB22_DisplayData".dbx15_7)) OR ("M30.5" AND "M10.4") OR "DB22_DisplayData".dbx14_2 OR "Reset" OR "ClampCutOk18" OR "V94_1") AND NOT "E16" AND NOT "Timer".T12.Q AND NOT "A30";
END_REGION

REGION Network 28: Forward on spool carriage(upward) and machine conveyor inverter
   RUNG wire#powerrail
      Contact( "Timer".T14.Q )
      Coil( "A13" )
   END_RUNG
   // the same network as SCL:
   "A13" := "Timer".T14.Q;
END_REGION

REGION Network 29: Backward on spool carriage(downward) and machine conveyor invert
   RUNG wire#powerrail
      Contact( "Timer".T19.Q )
      Coil( "A14" )
   END_RUNG
   // the same network as SCL:
   "A14" := "Timer".T19.Q;
END_REGION

REGION Network 30: Motor for spool carriage (Helix)
   RUNG wire#powerrail
      Contact( "Timer".T9.Q )
      Coil( "A20" )
   END_RUNG
   // the same network as SCL:
   "A20" := "Timer".T9.Q;
END_REGION

REGION Network 31: SUPPORT CALCULATION FOR SPOOL CARRIAGE MOVEMENT SPEED
   // Utilizzo DB3.DBW44 (diviso per 6) al posto di DB3.DBW46 per problemi dovuti al riavvio dopo EMG (se velocità tavola lenta, velocità carrello lentissima, a volte provoca fault inverter U221)
   RUNG wire#powerrail
      Div(in1 := "DB03_Machine".dbw44, in2 := 6, out => #wTemp)
   END_RUNG
   // the same network as SCL:
   #wTemp := "DB03_Machine".dbw44 / 6;
END_REGION

REGION Network 32
   // #DwTemp2
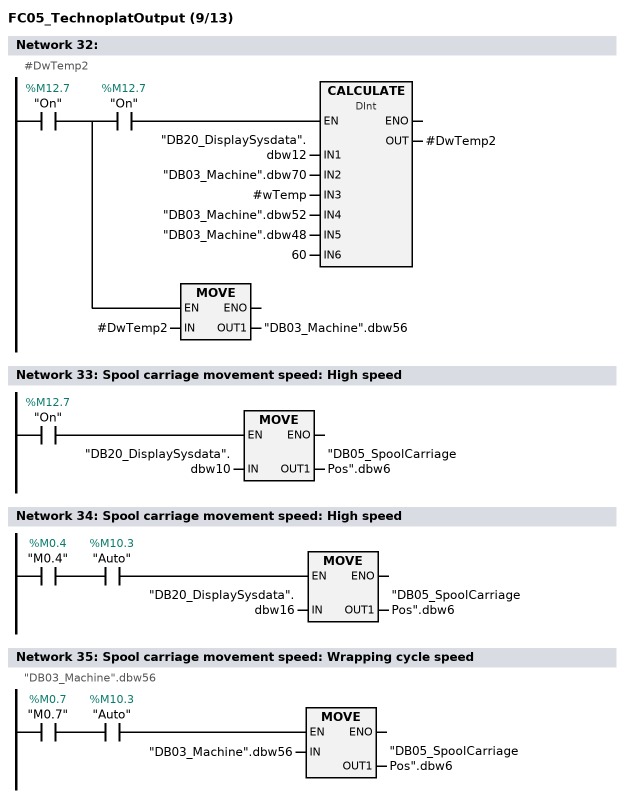
   RUNG wire#powerrail
      Contact( "On" )
      wire#w1
      Contact( "On" )
      { S7_Templates := "SrcType := DInt"; S7_GenerateENO := "TRUE"; S7_Expression := "((In1-In2)*In3*In4)/(In5*In6)" } Calculate(in1 := "DB20_DisplaySysdata".dbw12, in2 := "DB03_Machine".dbw70, in3 := #wTemp, in4 := "DB03_Machine".dbw52, in5 := "DB03_Machine".dbw48, in6 := 60, out => #DwTemp2)
   END_RUNG
   RUNG wire#w1
      { S7_GenerateENO := "TRUE" } Move(in := #DwTemp2, out1 => "DB03_Machine".dbw56)
   END_RUNG
   // the same network as SCL:
   IF "On" AND "On" THEN
       #DwTemp2 := (("DB20_DisplaySysdata".dbw12-"DB03_Machine".dbw70)*#wTemp*"DB03_Machine".dbw52)/("DB03_Machine".dbw48*60);
   END_IF;
   IF "On" THEN "DB03_Machine".dbw56 := #DwTemp2; END_IF;
END_REGION

REGION Network 33: Spool carriage movement speed: High speed
   RUNG wire#powerrail
      Contact( "On" )
      { S7_GenerateENO := "TRUE" } Move(in := "DB20_DisplaySysdata".dbw10, out1 => "DB05_SpoolCarriagePos".dbw6)
   END_RUNG
   // the same network as SCL:
   IF "On" THEN "DB05_SpoolCarriagePos".dbw6 := "DB20_DisplaySysdata".dbw10; END_IF;
END_REGION

REGION Network 34: Spool carriage movement speed: High speed
   RUNG wire#powerrail
      Contact( "M0.4" )
      Contact( "Auto" )
      { S7_GenerateENO := "TRUE" } Move(in := "DB20_DisplaySysdata".dbw16, out1 => "DB05_SpoolCarriagePos".dbw6)
   END_RUNG
   // the same network as SCL:
   IF "M0.4" AND "Auto" THEN "DB05_SpoolCarriagePos".dbw6 := "DB20_DisplaySysdata".dbw16; END_IF;
END_REGION

REGION Network 35: Spool carriage movement speed: Wrapping cycle speed
   // "DB03_Machine".dbw56
   RUNG wire#powerrail
      Contact( "M0.7" )
      Contact( "Auto" )
      { S7_GenerateENO := "TRUE" } Move(in := "DB03_Machine".dbw56, out1 => "DB05_SpoolCarriagePos".dbw6)
   END_RUNG
   // the same network as SCL:
   IF "M0.7" AND "Auto" THEN "DB05_SpoolCarriagePos".dbw6 := "DB03_Machine".dbw56; END_IF;
END_REGION

REGION Network 36: Spool carriage movement speed: Low speed
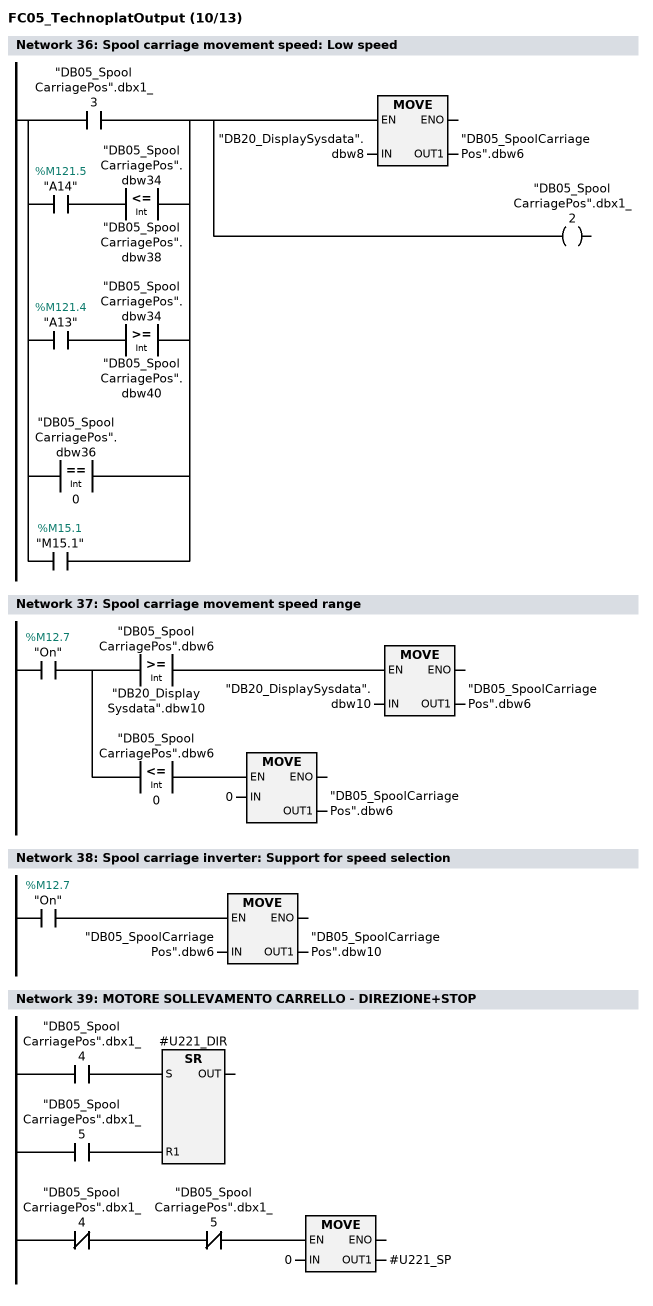
   RUNG wire#powerrail
      Contact( "DB05_SpoolCarriagePos".dbx1_3 )
      wire#w1
      { S7_GenerateENO := "TRUE" } Move(in := "DB20_DisplaySysdata".dbw8, out1 => "DB05_SpoolCarriagePos".dbw6)
   END_RUNG
   RUNG wire#powerrail
      Contact( "A14" )
      { S7_Templates := "SrcType := Int" } LE_Contact(in1 := "DB05_SpoolCarriagePos".dbw34, in2 := "DB05_SpoolCarriagePos".dbw38)
   END_RUNG wire#w1
   RUNG wire#powerrail
      Contact( "A13" )
      { S7_Templates := "SrcType := Int" } GE_Contact(in1 := "DB05_SpoolCarriagePos".dbw34, in2 := "DB05_SpoolCarriagePos".dbw40)
   END_RUNG wire#w1
   RUNG wire#powerrail
      { S7_Templates := "SrcType := Int" } EQ_Contact(in1 := "DB05_SpoolCarriagePos".dbw36, in2 := 0)
   END_RUNG wire#w1
   RUNG wire#powerrail
      Contact( "M15.1" )
   END_RUNG wire#w1
   RUNG wire#w1
      Coil( "DB05_SpoolCarriagePos".dbx1_2 )
   END_RUNG
   // the same network as SCL:
   #_w1 := "DB05_SpoolCarriagePos".dbx1_3 OR ("A14" AND ("DB05_SpoolCarriagePos".dbw34 <= "DB05_SpoolCarriagePos".dbw38)) OR ("A13" AND ("DB05_SpoolCarriagePos".dbw34 >= "DB05_SpoolCarriagePos".dbw40)) OR ("DB05_SpoolCarriagePos".dbw36 = 0) OR "M15.1";
   IF #_w1 THEN "DB05_SpoolCarriagePos".dbw6 := "DB20_DisplaySysdata".dbw8; END_IF;
   "DB05_SpoolCarriagePos".dbx1_2 := #_w1;
END_REGION

REGION Network 37: Spool carriage movement speed range
   RUNG wire#powerrail
      Contact( "On" )
      wire#w1
      { S7_Templates := "SrcType := Int" } GE_Contact(in1 := "DB05_SpoolCarriagePos".dbw6, in2 := "DB20_DisplaySysdata".dbw10)
      { S7_GenerateENO := "TRUE" } Move(in := "DB20_DisplaySysdata".dbw10, out1 => "DB05_SpoolCarriagePos".dbw6)
   END_RUNG
   RUNG wire#w1
      { S7_Templates := "SrcType := Int" } LE_Contact(in1 := "DB05_SpoolCarriagePos".dbw6, in2 := 0)
      { S7_GenerateENO := "TRUE" } Move(in := 0, out1 => "DB05_SpoolCarriagePos".dbw6)
   END_RUNG
   // the same network as SCL:
   IF "On" AND ("DB05_SpoolCarriagePos".dbw6 >= "DB20_DisplaySysdata".dbw10) THEN
       "DB05_SpoolCarriagePos".dbw6 := "DB20_DisplaySysdata".dbw10;
   END_IF;
   IF "On" AND ("DB05_SpoolCarriagePos".dbw6 <= 0) THEN "DB05_SpoolCarriagePos".dbw6 := 0; END_IF;
END_REGION

REGION Network 38: Spool carriage inverter: Support for speed selection
   RUNG wire#powerrail
      Contact( "On" )
      { S7_GenerateENO := "TRUE" } Move(in := "DB05_SpoolCarriagePos".dbw6, out1 => "DB05_SpoolCarriagePos".dbw10)
   END_RUNG
   // the same network as SCL:
   IF "On" THEN "DB05_SpoolCarriagePos".dbw10 := "DB05_SpoolCarriagePos".dbw6; END_IF;
END_REGION

REGION Network 39: MOTORE SOLLEVAMENTO CARRELLO - DIREZIONE+STOP
   RUNG wire#powerrail
      Contact( "DB05_SpoolCarriagePos".dbx1_4 )
      S_SR(operand := #U221_DIR, r1 := wire#w1)
   END_RUNG
   RUNG wire#powerrail
      Contact( "DB05_SpoolCarriagePos".dbx1_5 )
   END_RUNG wire#w1
   RUNG wire#powerrail
      I_Contact( "DB05_SpoolCarriagePos".dbx1_4 )
      I_Contact( "DB05_SpoolCarriagePos".dbx1_5 )
      Move(in := 0, out1 => #U221_SP)
   END_RUNG
   // the same network as SCL:
   IF "DB05_SpoolCarriagePos".dbx1_4 THEN
       #U221_DIR := TRUE;   // SR flip-flop
   END_IF;
   IF "DB05_SpoolCarriagePos".dbx1_5 THEN #U221_DIR := FALSE; END_IF;
   IF NOT "DB05_SpoolCarriagePos".dbx1_4 AND NOT "DB05_SpoolCarriagePos".dbx1_5 THEN #U221_SP := 0; END_IF;
END_REGION

REGION Network 40: MOTORE SOLLEVAMENTO CARRELLO - RIF.VELOCITA' + START
   // 2250 RPM = 75 HZ = 100% (3000@100HZ)
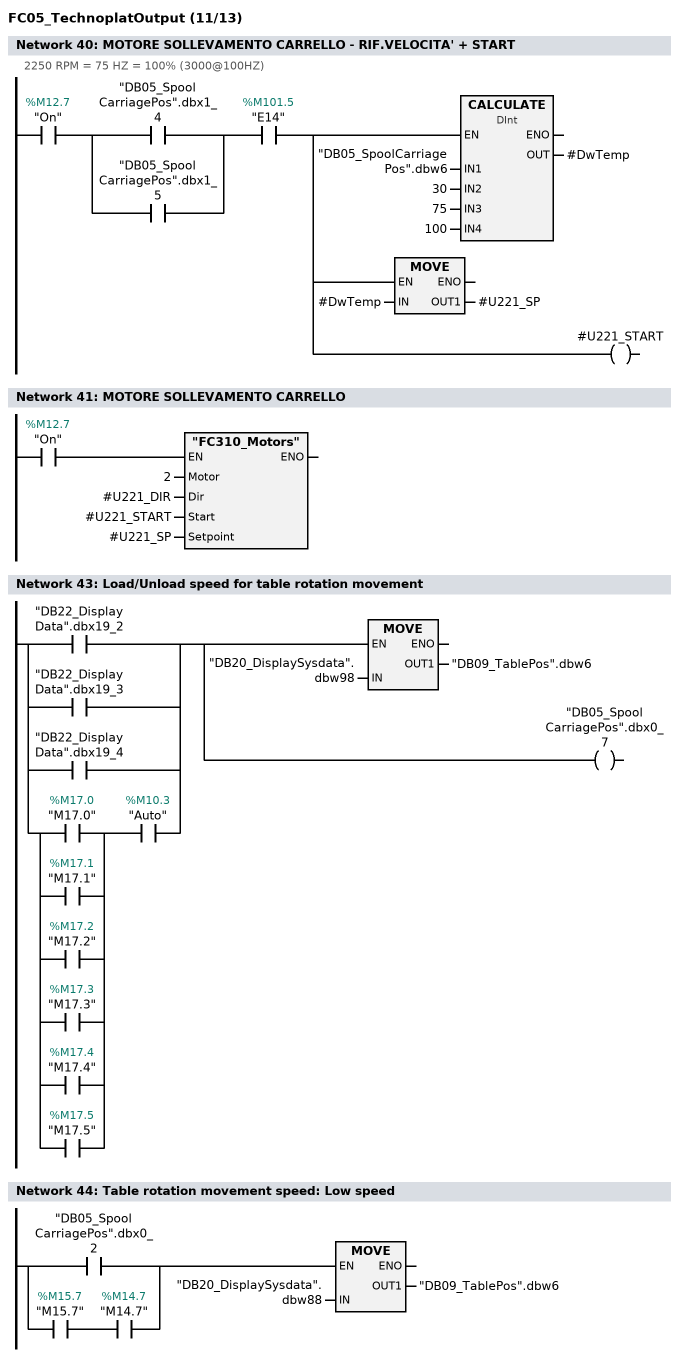
   RUNG wire#powerrail
      Contact( "On" )
      wire#w1
      Contact( "DB05_SpoolCarriagePos".dbx1_4 )
      wire#w2
      Contact( "E14" )
      wire#w3
      { S7_Templates := "SrcType := DInt"; S7_Expression := "(IN1*IN2*IN3)/IN4" } Calculate(in1 := "DB05_SpoolCarriagePos".dbw6, in2 := 30, in3 := 75, in4 := 100, out => #DwTemp)
   END_RUNG
   RUNG wire#w1
      Contact( "DB05_SpoolCarriagePos".dbx1_5 )
   END_RUNG wire#w2
   RUNG wire#w3
      Move(in := #DwTemp, out1 => #U221_SP)
   END_RUNG
   RUNG wire#w3
      Coil( #U221_START )
   END_RUNG
   // the same network as SCL:
   #_w1 := "On" AND ("DB05_SpoolCarriagePos".dbx1_4 OR "DB05_SpoolCarriagePos".dbx1_5) AND "E14";
   IF #_w1 THEN
       #DwTemp := ("DB05_SpoolCarriagePos".dbw6*30*75)/100;
       #U221_SP := #DwTemp;
   END_IF;
   #U221_START := #_w1;
END_REGION

REGION Network 41: MOTORE SOLLEVAMENTO CARRELLO
   RUNG wire#powerrail
      Contact( "On" )
      "FC310_Motors"(Motor := 2, Dir := #U221_DIR, Start := #U221_START, Setpoint := #U221_SP)
   END_RUNG
   // the same network as SCL:
   IF "On" THEN
       "FC310_Motors"(Motor := 2, Dir := #U221_DIR, Start := #U221_START, Setpoint := #U221_SP);
   END_IF;
END_REGION

REGION Network 42: Carriage and arm rotation speed conversion
END_REGION

REGION Network 43: Load/Unload speed for table rotation movement
   RUNG wire#powerrail
      Contact( "DB22_DisplayData".dbx19_2 )
      wire#w1
      { S7_GenerateENO := "TRUE" } Move(in := "DB20_DisplaySysdata".dbw98, out1 => "DB09_TablePos".dbw6)
   END_RUNG
   RUNG wire#powerrail
      Contact( "DB22_DisplayData".dbx19_3 )
   END_RUNG wire#w1
   RUNG wire#powerrail
      Contact( "DB22_DisplayData".dbx19_4 )
   END_RUNG wire#w1
   RUNG wire#powerrail
      Contact( "M17.0" )
      wire#w2
      Contact( "Auto" )
   END_RUNG wire#w1
   RUNG wire#powerrail
      Contact( "M17.1" )
   END_RUNG wire#w2
   RUNG wire#powerrail
      Contact( "M17.2" )
   END_RUNG wire#w2
   RUNG wire#powerrail
      Contact( "M17.3" )
   END_RUNG wire#w2
   RUNG wire#powerrail
      Contact( "M17.4" )
   END_RUNG wire#w2
   RUNG wire#powerrail
      Contact( "M17.5" )
   END_RUNG wire#w2
   RUNG wire#w1
      Coil( "DB05_SpoolCarriagePos".dbx0_7 )
   END_RUNG
   // the same network as SCL:
   #_w1 := "DB22_DisplayData".dbx19_2 OR "DB22_DisplayData".dbx19_3 OR "DB22_DisplayData".dbx19_4 OR (("M17.0" OR "M17.1" OR "M17.2" OR "M17.3" OR "M17.4" OR "M17.5") AND "Auto");
   IF #_w1 THEN "DB09_TablePos".dbw6 := "DB20_DisplaySysdata".dbw98; END_IF;
   "DB05_SpoolCarriagePos".dbx0_7 := #_w1;
END_REGION

REGION Network 44: Table rotation movement speed: Low speed
   RUNG wire#powerrail
      Contact( "DB05_SpoolCarriagePos".dbx0_2 )
      wire#w1
      { S7_GenerateENO := "TRUE" } Move(in := "DB20_DisplaySysdata".dbw88, out1 => "DB09_TablePos".dbw6)
   END_RUNG
   RUNG wire#powerrail
      Contact( "M15.7" )
      Contact( "M14.7" )
   END_RUNG wire#w1
   // the same network as SCL:
   IF "DB05_SpoolCarriagePos".dbx0_2 OR ("M15.7" AND "M14.7") THEN
       "DB09_TablePos".dbw6 := "DB20_DisplaySysdata".dbw88;
   END_IF;
END_REGION

REGION Network 45: EXTRA LOW
